             // Die Fehlerhaftigkeit des erkannten Parameter in der Fehlernummer eintragen   
             IF #piCount = 1 THEN
               #swParaError := #swParaError OR W#16#01;
             ELSIF #piCount = 2 THEN
               #swParaError := #swParaError OR W#16#02;
             ELSIF #piCount = 3 THEN
               #swParaError := #swParaError OR W#16#04;
             ELSIF #piCount = 4 THEN
               #swParaError := #swParaError OR W#16#08;
             ELSIF #piCount = 5 THEN
               #swParaError := #swParaError OR W#16#10;
             ELSIF #piCount = 6 THEN
               #swParaError := #swParaError OR W#16#20;
             ELSIF #piCount = 7 THEN
               #swParaError := #swParaError OR W#16#40;
             ELSIF #piCount = 8 THEN
               #swParaError := #swParaError OR W#16#80;
             ELSIF #piCount = 9 THEN
               #swParaError := #swParaError OR W#16#100;
             ELSIF #piCount = 10 THEN
               #swParaError := #swParaError OR W#16#200;
             ELSIF #piCount = 11 THEN
               #swParaError := #swParaError OR W#16#400;
             ELSIF #piCount = 12 THEN
               #swParaError := #swParaError OR W#16#800;
             ELSIF #piCount = 13 THEN
               #swParaError := #swParaError OR W#16#1000;
             ELSIF #piCount = 14 THEN
               #swParaError := #swParaError OR W#16#2000;
             ELSIF #piCount = 15 THEN
               #swParaError := #swParaError OR W#16#4000;
             ELSIF #piCount = #siParaNo THEN
               #swParaError := #swParaError OR W#16#8000;
             END_IF;

             // Zeiger auf nächsten Parametersatz setzen
             #piPointer := #piPointer + 6;

             // Format = Byte ? = > gesendeter Parameter ein Byte lang ohne Vorzeichen
           ELSIF (#sxRespParaMulti.sxData[#piPointer] = B#16#41) OR (#sxRespParaMulti.sxData[#piPointer] = B#16#05) THEN

             // ermittelter Parameterwert eintragen (Byte) 
             #sxParameter[#piCount].srValue := USINT_TO_REAL(BYTE_TO_USINT(#sxRespParaMulti.sxData[#piPointer + 2]));
             #sxParameter[#piCount].sdValue := 0;

             // ermittelte Fehlernummer im Puffer zurücksetzen
             #sxParameter[#piCount].swErrorNo := W#16#00;

             // Die Fehlerhaftigkeit des erkannten Parameter in der Fehlernummer löschen   
             IF #piCount = 1 THEN
               #swParaError := #swParaError AND W#16#FFFE;
             ELSIF #piCount = 2 THEN
               #swParaError := #swParaError AND W#16#FFFD;
             ELSIF #piCount = 3 THEN
               #swParaError := #swParaError AND W#16#FFFB;
             ELSIF #piCount = 4 THEN
               #swParaError := #swParaError AND W#16#FFF7;
             ELSIF #piCount = 5 THEN
               #swParaError := #swParaError AND W#16#FFEF;
             ELSIF #piCount = 6 THEN
               #swParaError := #swParaError AND W#16#FFDF;
             ELSIF #piCount = 7 THEN
               #swParaError := #swParaError AND W#16#FFBF;
             ELSIF #piCount = 8 THEN
               #swParaError := #swParaError AND W#16#FF7F;
             ELSIF #piCount = 9 THEN
               #swParaError := #swParaError AND W#16#FEFF;
             ELSIF #piCount = 10 THEN
               #swParaError := #swParaError AND W#16#FDFF;
             ELSIF #piCount = 11 THEN
               #swParaError := #swParaError AND W#16#FBFF;
             ELSIF #piCount = 12 THEN
               #swParaError := #swParaError AND W#16#F7FF;
             ELSIF #piCount = 13 THEN
               #swParaError := #swParaError AND W#16#EFFF;
             ELSIF #piCount = 14 THEN
               #swParaError := #swParaError AND W#16#DFFF;
             ELSIF #piCount = 15 THEN
               #swParaError := #swParaError AND W#16#BFFF;
             ELSIF #piCount = #siParaNo THEN
               #swParaError := #swParaError AND W#16#7FFF;
             END_IF;

             // Zeiger auf nächsten Parametersatz setzen
             #piPointer := #piPointer + 4;

             // Format = Byte ? = > gesendeter Parameter ein Byte lang mit Vorzeichen
           ELSIF (#sxRespParaMulti.sxData[#piPointer] = B#16#02) THEN

             // ermittelter Parameterwert eintragen (Byte) 
             #sxParameter[#piCount].srValue := SINT_TO_REAL(BYTE_TO_SINT(#sxRespParaMulti.sxData[#piPointer + 2]));
             #sxParameter[#piCount].sdValue := 0;

             // ermittelte Fehlernummer im Puffer zurücksetzen
             #sxParameter[#piCount].swErrorNo := W#16#00;

             // Die Fehlerhaftigkeit des erkannten Parameter in der Fehlernummer löschen   
             IF #piCount = 1 THEN
               #swParaError := #swParaError AND W#16#FFFE;
             ELSIF #piCount = 2 THEN
               #swParaError := #swParaError AND W#16#FFFD;
             ELSIF #piCount = 3 THEN
               #swParaError := #swParaError AND W#16#FFFB;
             ELSIF #piCount = 4 THEN
               #swParaError := #swParaError AND W#16#FFF7;
             ELSIF #piCount = 5 THEN
               #swParaError := #swParaError AND W#16#FFEF;
             ELSIF #piCount = 6 THEN
               #swParaError := #swParaError AND W#16#FFDF;
             ELSIF #piCount = 7 THEN
               #swParaError := #swParaError AND W#16#FFBF;
             ELSIF #piCount = 8 THEN
               #swParaError := #swParaError AND W#16#FF7F;
             ELSIF #piCount = 9 THEN
               #swParaError := #swParaError AND W#16#FEFF;
             ELSIF #piCount = 10 THEN
               #swParaError := #swParaError AND W#16#FDFF;
             ELSIF #piCount = 11 THEN
               #swParaError := #swParaError AND W#16#FBFF;
             ELSIF #piCount = 12 THEN
               #swParaError := #swParaError AND W#16#F7FF;
             ELSIF #piCount = 13 THEN
               #swParaError := #swParaError AND W#16#EFFF;
             ELSIF #piCount = 14 THEN
               #swParaError := #swParaError AND W#16#DFFF;
             ELSIF #piCount = 15 THEN
               #swParaError := #swParaError AND W#16#BFFF;
             ELSIF #piCount = #siParaNo THEN
               #swParaError := #swParaError AND W#16#7FFF;
             END_IF;

             // Zeiger auf nächsten Parametersatz setzen
             #piPointer := #piPointer + 4;

             // Format = Word ? = > gesendeter Parameter zwei Bytes lang ohne Vorzeichen
           ELSIF (#sxRespParaMulti.sxData[#piPointer] = B#16#42) OR (#sxRespParaMulti.sxData[#piPointer] = B#16#06)
             OR (#sxRespParaMulti.sxData[#piPointer] = B#16#0A) THEN

             // Format = Word, zwei Bytes zu übermitteltem Parameterwert zusammenfassen
             #pwWordHigh := SHL(IN := BYTE_TO_WORD(#sxRespParaMulti.sxData[#piPointer + 2]), N := 8);
             #pwWordLow := BYTE_TO_WORD(#sxRespParaMulti.sxData[#piPointer + 3]);
             #pwWord1 := #pwWordHigh XOR #pwWordLow;

             // ermittelter Parameterwert eintragen (Word)
             #sxParameter[#piCount].srValue := UINT_TO_REAL(WORD_TO_UINT(#pwWord1));
             #sxParameter[#piCount].sdValue := 0;

             // ermittelte Fehlernummer im Puffer zurücksetzen
             #sxParameter[#piCount].swErrorNo := W#16#00;

             // Die Fehlerhaftigkeit des erkannten Parameter in der Fehlernummer löschen   
             IF #piCount = 1 THEN
               #swParaError := #swParaError AND W#16#FFFE;
             ELSIF #piCount = 2 THEN
               #swParaError := #swParaError AND W#16#FFFD;
             ELSIF #piCount = 3 THEN
               #swParaError := #swParaError AND W#16#FFFB;
             ELSIF #piCount = 4 THEN
               #swParaError := #swParaError AND W#16#FFF7;
             ELSIF #piCount = 5 THEN
               #swParaError := #swParaError AND W#16#FFEF;
             ELSIF #piCount = 6 THEN
               #swParaError := #swParaError AND W#16#FFDF;
             ELSIF #piCount = 7 THEN
               #swParaError := #swParaError AND W#16#FFBF;
             ELSIF #piCount = 8 THEN
               #swParaError := #swParaError AND W#16#FF7F;
             ELSIF #piCount = 9 THEN
               #swParaError := #swParaError AND W#16#FEFF;
             ELSIF #piCount = 10 THEN
               #swParaError := #swParaError AND W#16#FDFF;
             ELSIF #piCount = 11 THEN
               #swParaError := #swParaError AND W#16#FBFF;
             ELSIF #piCount = 12 THEN
               #swParaError := #swParaError AND W#16#F7FF;
             ELSIF #piCount = 13 THEN
               #swParaError := #swParaError AND W#16#EFFF;
             ELSIF #piCount = 14 THEN
               #swParaError := #swParaError AND W#16#DFFF;
             ELSIF #piCount = 15 THEN
               #swParaError := #swParaError AND W#16#BFFF;
             ELSIF #piCount = #siParaNo THEN
               #swParaError := #swParaError AND W#16#7FFF;
             END_IF;

             // Zeiger auf nächsten Parametersatz setzen
             #piPointer := #piPointer + 4;

             // Format = Word ? = > gesendeter Parameter zwei Bytes lang mit Vorzeichen
           ELSIF (#sxRespParaMulti.sxData[#piPointer] = B#16#03) THEN

             // Format = Word, zwei Bytes zu übermitteltem Parameterwert zusammenfassen
             #pwWordHigh := SHL(IN := BYTE_TO_WORD(#sxRespParaMulti.sxData[#piPointer + 2]), N := 8);
             #pwWordLow := BYTE_TO_WORD(#sxRespParaMulti.sxData[#piPointer + 3]);
             #pwWord1 := #pwWordHigh XOR #pwWordLow;

             // ermittelter Parameterwert eintragen (Word)
             #sxParameter[#piCount].srValue := INT_TO_REAL(WORD_TO_INT(#pwWord1));
             #sxParameter[#piCount].sdValue := 0;

             // ermittelte Fehlernummer im Puffer zurücksetzen
             #sxParameter[#piCount].swErrorNo := W#16#00;

             // Die Fehlerhaftigkeit des erkannten Parameter in der Fehlernummer löschen   
             IF #piCount = 1 THEN
               #swParaError := #swParaError AND W#16#FFFE;
             ELSIF #piCount = 2 THEN
               #swParaError := #swParaError AND W#16#FFFD;
             ELSIF #piCount = 3 THEN
               #swParaError := #swParaError AND W#16#FFFB;
             ELSIF #piCount = 4 THEN
               #swParaError := #swParaError AND W#16#FFF7;
             ELSIF #piCount = 5 THEN
               #swParaError := #swParaError AND W#16#FFEF;
             ELSIF #piCount = 6 THEN
               #swParaError := #swParaError AND W#16#FFDF;
             ELSIF #piCount = 7 THEN
               #swParaError := #swParaError AND W#16#FFBF;
             ELSIF #piCount = 8 THEN
               #swParaError := #swParaError AND W#16#FF7F;
             ELSIF #piCount = 9 THEN
               #swParaError := #swParaError AND W#16#FEFF;
             ELSIF #piCount = 10 THEN
               #swParaError := #swParaError AND W#16#FDFF;
             ELSIF #piCount = 11 THEN
               #swParaError := #swParaError AND W#16#FBFF;
             ELSIF #piCount = 12 THEN
               #swParaError := #swParaError AND W#16#F7FF;
             ELSIF #piCount = 13 THEN
               #swParaError := #swParaError AND W#16#EFFF;
             ELSIF #piCount = 14 THEN
               #swParaError := #swParaError AND W#16#DFFF;
             ELSIF #piCount = 15 THEN
               #swParaError := #swParaError AND W#16#BFFF;
             ELSIF #piCount = #siParaNo THEN
               #swParaError := #swParaError AND W#16#7FFF;
             END_IF;

             // Zeiger auf nächsten Parametersatz setzen
             #piPointer := #piPointer + 4;

             // Format = Double Word ? = > gesendeter Parameter vier Bytes lang ohne Vorzeichen
           ELSIF (#sxRespParaMulti.sxData[#piPointer] = B#16#43) OR (#sxRespParaMulti.sxData[#piPointer] = B#16#07) OR
             (#sxRespParaMulti.sxData[#piPointer] = B#16#0D) THEN

             // Format = Double Word, vier Bytes zu übermitteltem Parameterwert zusammenfassen
             #pwWordHigh := SHL(IN := BYTE_TO_WORD(#sxRespParaMulti.sxData[#piPointer + 2]), N := 8);
             #pwWordLow := BYTE_TO_WORD(#sxRespParaMulti.sxData[#piPointer + 3]);
             #pwWord1 := #pwWordHigh XOR #pwWordLow;

             #pwWordHigh := SHL(IN := BYTE_TO_WORD(#sxRespParaMulti.sxData[#piPointer + 4]), N := 8);
             #pwWordLow := BYTE_TO_WORD(#sxRespParaMulti.sxData[#piPointer + 5]);
             #pwWord2 := #pwWordHigh XOR #pwWordLow;

             #pdDWordHigh := SHL(IN := WORD_TO_DWORD(#pwWord1), N := 16);
             #pdDWordLow := WORD_TO_DWORD(#pwWord2);

             // ermittelter Parameterwert eintragen (Word)
             #sxParameter[#piCount].srValue := 0.0;
             #sxParameter[#piCount].sdValue := DWORD_TO_DINT(#pdDWordHigh XOR #pdDWordLow);

             // ermittelte Fehlernummer im Puffer zurücksetzen
             #sxParameter[#piCount].swErrorNo := W#16#00;

             // Die Fehlerhaftigkeit des erkannten Parameter in der Fehlernummer löschen   
             IF #piCount = 1 THEN
               #swParaError := #swParaError AND W#16#FFFE;
             ELSIF #piCount = 2 THEN
               #swParaError := #swParaError AND W#16#FFFD;
             ELSIF #piCount = 3 THEN
               #swParaError := #swParaError AND W#16#FFFB;
             ELSIF #piCount = 4 THEN
               #swParaError := #swParaError AND W#16#FFF7;
             ELSIF #piCount = 5 THEN
               #swParaError := #swParaError AND W#16#FFEF;
             ELSIF #piCount = 6 THEN
               #swParaError := #swParaError AND W#16#FFDF;
             ELSIF #piCount = 7 THEN
               #swParaError := #swParaError AND W#16#FFBF;
             ELSIF #piCount = 8 THEN
               #swParaError := #swParaError AND W#16#FF7F;
             ELSIF #piCount = 9 THEN
               #swParaError := #swParaError AND W#16#FEFF;
             ELSIF #piCount = 10 THEN
               #swParaError := #swParaError AND W#16#FDFF;
             ELSIF #piCount = 11 THEN
               #swParaError := #swParaError AND W#16#FBFF;
             ELSIF #piCount = 12 THEN
               #swParaError := #swParaError AND W#16#F7FF;
             ELSIF #piCount = 13 THEN
               #swParaError := #swParaError AND W#16#EFFF;
             ELSIF #piCount = 14 THEN
               #swParaError := #swParaError AND W#16#DFFF;
             ELSIF #piCount = 15 THEN
               #swParaError := #swParaError AND W#16#BFFF;
             ELSIF #piCount = #siParaNo THEN
               #swParaError := #swParaError AND W#16#7FFF;
             END_IF;

             // Zeiger auf nächsten Parametersatz setzen
             #piPointer := #piPointer + 6;

             // Format = Double Word ? = > gesendeter Parameter vier Bytes lang mit Vorzeichen
           ELSIF (#sxRespParaMulti.sxData[#piPointer] = B#16#04) THEN

             // Format = Double Word, vier Bytes zu übermitteltem Parameterwert zusammenfassen
             #pwWordHigh := SHL(IN := BYTE_TO_WORD(#sxRespParaMulti.sxData[#piPointer + 2]), N := 8);
             #pwWordLow := BYTE_TO_WORD(#sxRespParaMulti.sxData[#piPointer + 3]);
             #pwWord1 := #pwWordHigh XOR #pwWordLow;

             #pwWordHigh := SHL(IN := BYTE_TO_WORD(#sxRespParaMulti.sxData[#piPointer + 4]), N := 8);
             #pwWordLow := BYTE_TO_WORD(#sxRespParaMulti.sxData[#piPointer + 5]);
             #pwWord2 := #pwWordHigh XOR #pwWordLow;

             #pdDWordHigh := SHL(IN := WORD_TO_DWORD(#pwWord1), N := 16);
             #pdDWordLow := WORD_TO_DWORD(#pwWord2);

             // ermittelter Parameterwert eintragen (Word)
             #sxParameter[#piCount].srValue := 0.0;
             #sxParameter[#piCount].sdValue := DWORD_TO_DINT(#pdDWordHigh XOR #pdDWordLow);

             // ermittelte Fehlernummer im Puffer zurücksetzen
             #sxParameter[#piCount].swErrorNo := W#16#00;

             // Die Fehlerhaftigkeit des erkannten Parameter in der Fehlernummer löschen   
             IF #piCount = 1 THEN
               #swParaError := #swParaError AND W#16#FFFE;
             ELSIF #piCount = 2 THEN
               #swParaError := #swParaError AND W#16#FFFD;
             ELSIF #piCount = 3 THEN
               #swParaError := #swParaError AND W#16#FFFB;
             ELSIF #piCount = 4 THEN
               #swParaError := #swParaError AND W#16#FFF7;
             ELSIF #piCount = 5 THEN
               #swParaError := #swParaError AND W#16#FFEF;
             ELSIF #piCount = 6 THEN
               #swParaError := #swParaError AND W#16#FFDF;
             ELSIF #piCount = 7 THEN
               #swParaError := #swParaError AND W#16#FFBF;
             ELSIF #piCount = 8 THEN
               #swParaError := #swParaError AND W#16#FF7F;
             ELSIF #piCount = 9 THEN
               #swParaError := #swParaError AND W#16#FEFF;
             ELSIF #piCount = 10 THEN
               #swParaError := #swParaError AND W#16#FDFF;
             ELSIF #piCount = 11 THEN
               #swParaError := #swParaError AND W#16#FBFF;
             ELSIF #piCount = 12 THEN
               #swParaError := #swParaError AND W#16#F7FF;
             ELSIF #piCount = 13 THEN
               #swParaError := #swParaError AND W#16#EFFF;
             ELSIF #piCount = 14 THEN
               #swParaError := #swParaError AND W#16#DFFF;
             ELSIF #piCount = 15 THEN
               #swParaError := #swParaError AND W#16#BFFF;
             ELSIF #piCount = #siParaNo THEN
               #swParaError := #swParaError AND W#16#7FFF;
             END_IF;

             // Zeiger auf nächsten Parametersatz setzen
             #piPointer := #piPointer + 6;

             // Format = Double Word ? = > gesendeter Parameter vier Bytes lang (FloatingPoint)
           ELSIF (#sxRespParaMulti.sxData[#piPointer] = B#16#08) THEN

             // Format = Double Word, vier Bytes zu übermitteltem Parameterwert zusammenfassen
             #pwWordHigh := SHL(IN := BYTE_TO_WORD(#sxRespParaMulti.sxData[#piPointer + 2]), N := 8);
             #pwWordLow := BYTE_TO_WORD(#sxRespParaMulti.sxData[#piPointer + 3]);
             #pwWord1 := #pwWordHigh XOR #pwWordLow;

             #pwWordHigh := SHL(IN := BYTE_TO_WORD(#sxRespParaMulti.sxData[#piPointer + 4]), N := 8);
             #pwWordLow := BYTE_TO_WORD(#sxRespParaMulti.sxData[#piPointer + 5]);
             #pwWord2 := #pwWordHigh XOR #pwWordLow;

             #pdDWordHigh := SHL(IN := WORD_TO_DWORD(#pwWord1), N := 16);
             #pdDWordLow := WORD_TO_DWORD(#pwWord2);

             // ermittelter Parameterwert eintragen (Word)
             #sxParameter[#piCount].srValue := DWORD_TO_REAL(#pdDWordHigh XOR #pdDWordLow);
             #sxParameter[#piCount].sdValue := 0;

             // ermittelte Fehlernummer im Puffer zurücksetzen
             #sxParameter[#piCount].swErrorNo := W#16#00;

             // Die Fehlerhaftigkeit des erkannten Parameter in der Fehlernummer löschen   
             IF #piCount = 1 THEN
               #swParaError := #swParaError AND W#16#FFFE;
             ELSIF #piCount = 2 THEN
               #swParaError := #swParaError AND W#16#FFFD;
             ELSIF #piCount = 3 THEN
               #swParaError := #swParaError AND W#16#FFFB;
             ELSIF #piCount = 4 THEN
               #swParaError := #swParaError AND W#16#FFF7;
             ELSIF #piCount = 5 THEN
               #swParaError := #swParaError AND W#16#FFEF;
             ELSIF #piCount = 6 THEN
               #swParaError := #swParaError AND W#16#FFDF;
             ELSIF #piCount = 7 THEN
               #swParaError := #swParaError AND W#16#FFBF;
             ELSIF #piCount = 8 THEN
               #swParaError := #swParaError AND W#16#FF7F;
             ELSIF #piCount = 9 THEN
               #swParaError := #swParaError AND W#16#FEFF;
             ELSIF #piCount = 10 THEN
               #swParaError := #swParaError AND W#16#FDFF;
             ELSIF #piCount = 11 THEN
               #swParaError := #swParaError AND W#16#FBFF;
             ELSIF #piCount = 12 THEN
               #swParaError := #swParaError AND W#16#F7FF;
             ELSIF #piCount = 13 THEN
               #swParaError := #swParaError AND W#16#EFFF;
             ELSIF #piCount = 14 THEN
               #swParaError := #swParaError AND W#16#DFFF;
             ELSIF #piCount = 15 THEN
               #swParaError := #swParaError AND W#16#BFFF;
             ELSIF #piCount = #siParaNo THEN
               #swParaError := #swParaError AND W#16#7FFF;
             END_IF;

             // Zeiger auf nächsten Parametersatz setzen
             #piPointer := #piPointer + 6;

             // Unbekanter Datentyp
           ELSE

             #siErrorId := 5;
             #sbError := True;
             #sbDone := False;
             // Die Fehlerhaftigkeit des erkannten Parameter in der Fehlernummer eintragen   
             IF #piCount = 1 THEN
               #swParaError := #swParaError OR W#16#01;
             ELSIF #piCount = 2 THEN
               #swParaError := #swParaError OR W#16#02;
             ELSIF #piCount = 3 THEN
               #swParaError := #swParaError OR W#16#04;
             ELSIF #piCount = 4 THEN
               #swParaError := #swParaError OR W#16#08;
             ELSIF #piCount = 5 THEN
               #swParaError := #swParaError OR W#16#10;
             ELSIF #piCount = 6 THEN
               #swParaError := #swParaError OR W#16#20;
             ELSIF #piCount = 7 THEN
               #swParaError := #swParaError OR W#16#40;
             ELSIF #piCount = 8 THEN
               #swParaError := #swParaError OR W#16#80;
             ELSIF #piCount = 9 THEN
               #swParaError := #swParaError OR W#16#100;
             ELSIF #piCount = 10 THEN
               #swParaError := #swParaError OR W#16#200;
             ELSIF #piCount = 11 THEN
               #swParaError := #swParaError OR W#16#400;
             ELSIF #piCount = 12 THEN
               #swParaError := #swParaError OR W#16#800;
             ELSIF #piCount = 13 THEN
               #swParaError := #swParaError OR W#16#1000;
             ELSIF #piCount = 14 THEN
               #swParaError := #swParaError OR W#16#2000;
             ELSIF #piCount = 15 THEN
               #swParaError := #swParaError OR W#16#4000;
             ELSIF #piCount = #siParaNo THEN
               #swParaError := #swParaError OR W#16#8000;
             END_IF;

             EXIT; //Bei erstem unbekannten Datentyp abrechen

           END_IF;
         END_FOR; // die angefragten Parameter auswerten und im Puffer abspeichern

         // Fehlerkennung zurücknehmen
         IF (#siErrorId = 3) OR (#siErrorId = 1) THEN
           #siErrorId := 0;
           #sbError := False;
         END_IF;

         #DiagId := W#16#00;

         // Auftrag : Parameter lesen ist abgeschlossen
         #sbRdStart := False;
         #sbRead := False;
       END_IF; // kein Fehler beim LESEN AZYKLISCH und Auftrag fertig 
     END_IF; // vom Auftrag "Parameter lesen" die Antwort abwarten und dann auswerten
   END_IF; // Auftrag "Parameter lesen" wurde ausgelöst


   // Auftrag "Parameter schreiben" wurde ausgelöst
   IF #sbParaNo AND NOT #sbRead AND #sbWrite THEN

     // Auftrag "Parameter schreiben" bzw. "ändern" besteht aus zwei Aufträgen
     // 1. Teilauftrag "Parameter lesen"
     // 2. Teilauftrag "Parameter schreiben bzw. ändern"

     // 1. Teilauftrag "Parameter lesen" vorbereiten und abschicken
     IF #sbWrStart1 THEN

       // Ablöschen des Sendepuffers
       IF NOT (#siParaNo = #siParaNoMax) THEN
         FOR #piCount := #siParaNo TO #siParaNoMax DO

           // Parameternummer des Parameters 
           #sxReqParaMulti.sxParaAdress[#piCount].siParaNo := 0;

           // Subindex des Parameters
           #sxReqParaMulti.sxParaAdress[#piCount].siIndex := 0;
         END_FOR;
       END_IF;

       // Auftrags-HEADER erstellen
       // Auftragsreferenz
       #sxReqParaMulti.sxHeader.syReqRef := INT_TO_BYTE(#siReqRef);

       // Auftragskennung 0x01=Request Parameters
       #sxReqParaMulti.sxHeader.syReqId := B#16#01;

       // Achse
       #sxReqParaMulti.sxHeader.syAxisNo := #syAxisNo;

       // Anzahl Parameter        
       #sxReqParaMulti.sxHeader.syParaNo := INT_TO_BYTE(#siParaNo);

       // Auftrags-PARAMETERADRESSE erstellen
       FOR #piCount := 1 TO #siParaNo DO

         // Parameternummer des Parameters                                
         #sxReqParaMulti.sxParaAdress[#piCount].siParaNo := #sxParameter[#piCount].siParaNo;

         // Subindex des Parameters
         #sxReqParaMulti.sxParaAdress[#piCount].siIndex := #sxParameter[#piCount].siIndex;
       END_FOR;

       // SCHREIBEN AZYKLISCH
       #piLenTele := #siLenHeader + #siLenParaMulti;
       #WRREC_1(REQ := True,                                // Startimpuls
                ID := #hardwareId,                         // Diagnoseadresse
                INDEX := 47,                                  // Rahmentyp
                LEN := INT_TO_UINT(#piLenTele),             // maximale Länge
                DONE => #sbWrDone,                           // Schreibauftrag beendet
                BUSY => #sbWrBusy,                           // Slave beschäftigt
                ERROR => #sbWrError,                          // Fehler beim Schreiben
                STATUS => #pdStatus,                           // Status[1] = Error => Status[2] Error Decode + Status[3] Error Code
                RECORD := #sxReqParaMulti);                    // Zeiger auf zu schreibenen Datensatz

       // Ausgänge setzen
       #sbBusy := #sbWrBusy;
       #sbDone := #sbWrDone;

       // Fehler auswerten
       IF #sbWrError THEN

         // Fehlerstatus aus dem Doppelwort filtern und weitergeben                
         #pwWord1 := DWORD_TO_WORD(SHR(IN := (#pdStatus AND DW#16#FFFF00), N := 8));

         // Fehlerstatus setzen
         #siErrorId := 3;
         #DiagId := #pwWord1;

         //Temporärer Fehler: #pdStatus = 80A7, 80B5, 80C0, 80C1, 80C2, 80C3 oder 80C4 zulassen und nocheinmal versuchen
         IF NOT (#pwWord1 = DW#16#80A7) AND NOT (#pwWord1 = DW#16#80B5) AND NOT (#pwWord1 = DW#16#80C0) AND
           NOT (#pwWord1 = DW#16#80C1) AND NOT (#pwWord1 = DW#16#80C2) AND NOT (#pwWord1 = DW#16#80C3) AND
           NOT (#pwWord1 = DW#16#80C4) THEN

           // Wiederholungsauftrag wieder zurücknehmen
           #sbWrStart1 := False;
           #sbRdStart1 := False;
           #sbWrite := False;

           // Fehler ausgeben 
           #sbError := #sbWrError;

         ELSE
           // Fehlerwiederholauftrag ??                   
           IF #siErrorCount = #siMaxErrCount THEN

             // Wiederholungsauftrag wieder zurücknehmen
             #sbWrStart1 := False;
             #sbRdStart1 := False;
             #sbWrite := False;

             //Fehlerzähler zurücksetzen
             #siErrorCount := 0;

             // Fehler ausgeben 
             #sbError := #sbWrError;

             // nix tun bis Zähler überläuft
           ELSE
             #siErrorCount := #siErrorCount + 1;
           END_IF;
         END_IF;

         // kein Fehler beim SCHEIBEN AZYKLISCH und Auftrag fertig 
       ELSIF NOT #sbWrBusy AND #sbWrDone THEN

         // Fehlerkennung zurücknehmen
         IF (#siErrorId = 3) THEN
           #siErrorId := 0;
           #sbError := False;
         END_IF;

         #DiagId := W#16#00;

         // Schreibauftrag fertig melden und Leseantrag anstossen
         #sbWrStart1 := False;
         #sbRdStart1 := True;
       END_IF;
     END_IF; // 1. Teilauftrag "Parameter lesen" vorbereiten und abschicken

     // vom 1. Teilauftrag "Parameter lesen" die Antwort abwarten und dann auswerten
     IF #sbRdStart1 THEN

       // Ablöschen des Empfangspuffers
       #sxRespParaMulti.sxHeader.syReqRef := B#16#00;
       #sxRespParaMulti.sxHeader.syReqId := B#16#00;
       #sxRespParaMulti.sxHeader.syAxisNo := B#16#00;
       #sxRespParaMulti.sxHeader.syParaNo := B#16#00;

       FOR #piCount := 1 TO #siLenParaMulti DO
         #sxRespParaMulti.sxData[#piCount] := B#16#00;
       END_FOR;

       // LESEN AZYKLISCH
       #piLenTele := #siLenHeader + #siLenParaMulti;
       #RDREC_1(REQ := True,                                // Startimpuls
                ID := #hardwareId,                         // Diagnoseadresse        
                INDEX := 47,                                  // Rahmentyp           
                MLEN := INT_TO_UINT(#piLenTele),             // maximale Länge
                VALID => #pbValidSFB,                         // neuer Datensatz empfangen und gültig      
                BUSY => #sbRdBusy,                           // Slave beschäftigt
                ERROR => #sbRdError,                          // Fehler beim Schreiben
                STATUS => #pdStatus,                           // Status[1] = Error => Status[2] Error Decode + Status[3] Error Code 
                LEN => #piLenSFB,                           // Länge des gelesenen Datensatzes
                RECORD := #sxRespParaMulti);                   // Zeiger auf gelesenen Datensatz

       // Ausgänge setzen
       #sbBusy := #sbRdBusy;
       #sbDone := #pbValidSFB;

       // Fehler auswerten
       IF #sbRdError THEN
         // Fehlerstatus aus dem Doppelwort filtern und weitergeben                
         #pwWord1 := DWORD_TO_WORD(SHR(IN := (#pdStatus AND DW#16#FFFF00), N := 8));

         // Fehlerstatus setzen
         #siErrorId := 3;
         #DiagId := #pwWord1;

         //Temporärer Fehler: #pdStatus = 80A7, 80B5, 80C0, 80C1, 80C2, 80C3 oder 80C4 zulassen und nocheinmal versuchen
         IF NOT (#pwWord1 = DW#16#80A7) AND NOT (#pwWord1 = DW#16#80B5) AND NOT (#pwWord1 = DW#16#80C0) AND
           NOT (#pwWord1 = DW#16#80C1) AND NOT (#pwWord1 = DW#16#80C2) AND NOT (#pwWord1 = DW#16#80C3) AND
           NOT (#pwWord1 = DW#16#80C4) THEN

           // Wiederholungsauftrag wieder zurücknehmen
           #sbWrStart1 := False;
           #sbRdStart1 := False;
           #sbWrite := False;

           // Fehler ausgeben 
           #sbError := #sbRdError;

         ELSE
           // Fehlerwiederholauftrag ??                   
           IF #siErrorCount = #siMaxErrCount THEN

             // Wiederholungsauftrag wieder zurücknehmen
             #sbWrStart1 := False;
             #sbRdStart1 := False;
             #sbWrite := False;

             //Fehlerzähler zurücksetzen
             #siErrorCount := 0;

             // Fehler ausgeben 
             #sbError := #sbRdError;

             // nix tun bis Zähler überläuft
           ELSE
             #siErrorCount := #siErrorCount + 1;
           END_IF;
         END_IF;

         // Fehler : die Auftragsreferenz der Antwort übertimmt nicht mit der Auftragsreferenz der Anfrage überein
       ELSIF NOT (#siReqRef = BYTE_TO_INT(#sxRespParaMulti.sxHeader.syReqRef)) AND NOT #sbRdBusy AND #pbValidSFB THEN
         #siErrorId := 1;
         #sbError := True;
         #sbDone := False;

         // Wiederholungsauftrag wieder zurücknehmen
         #sbWrStart1 := False;
         #sbRdStart1 := False;
         #sbWrite := False;

         // Fehler : falsche Auftragskennung zurück erhalten    
       ELSIF NOT (#sxRespParaMulti.sxHeader.syReqId = B#16#81 OR #sxRespParaMulti.sxHeader.syReqId = B#16#01) AND
         NOT #sbRdBusy AND #pbValidSFB THEN
         #siErrorId := 1;
         #sbError := True;
         #sbDone := False;

         // Wiederholungsauftrag wieder zurücknehmen
         #sbWrStart1 := False;
         #sbRdStart1 := False;
         #sbWrite := False;

         // Fehler : die angeforderte Anzahl Parameter entspricht nicht der übermittelten Anzahl Parameter überein
       ELSIF NOT (#siParaNo = BYTE_TO_INT(#sxRespParaMulti.sxHeader.syParaNo)) AND NOT #sbRdBusy AND #pbValidSFB THEN
         #siErrorId := 1;
         #sbError := True;
         #sbDone := False;

         // Wiederholungsauftrag wieder zurücknehmen
         #sbWrStart1 := False;
         #sbRdStart1 := False;
         #sbWrite := False;

         // Fehler : die Achse entspricht nicht der übergebenen Achse
       ELSIF NOT (#syAxisNo = #sxRespParaMulti.sxHeader.syAxisNo) AND NOT #sbRdBusy AND #pbValidSFB THEN
         #siErrorId := 1;
         #sbError := True;
         #sbDone := False;

         // Wiederholungsauftrag wieder zurücknehmen
         #sbWrStart1 := False;
         #sbRdStart1 := False;
         #sbWrite := False;

         // kein Fehler beim LESEN AZYKLISCH und Auftrag fertig 
       ELSIF NOT #sbRdBusy AND #pbValidSFB THEN

         // die angefragten Parameter auswerten und im Puffer abspeichern
         #piPointer := 1;
         #swParaError := 16#0;

         FOR #piCount := 1 TO #siParaNo DO

           // ermitteltes Format des Parameters abspeichern
           #sxParameter[#piCount].syFormat := #sxRespParaMulti.sxData[#piPointer];

           // Format = Error ? = > gesendeter Parameter fehlerhaft
           IF (BYTE_TO_INT(#sxRespParaMulti.sxData[#piPointer]) = 68) THEN

             // Format = Error, zwei Bytes zu übermittelten Fehlernummer zusammenfassen
             #pwWordHigh := SHL(IN := BYTE_TO_WORD(#sxRespParaMulti.sxData[#piPointer + 2]), N := 8);
             #pwWordLow := BYTE_TO_WORD(#sxRespParaMulti.sxData[#piPointer + 3]);

             #sbError := True;

             // ermittelte Fehlernummer im Puffer abspeichern
             #sxParameter[#piCount].swErrorNo := #pwWordHigh XOR #pwWordLow;

             // Die Fehlerhaftigkeit des erkannten Parameter in der Fehlernummer eintragen   
             IF #piCount = 1 THEN
               #swParaError := #swParaError OR W#16#01;
             ELSIF #piCount = 2 THEN
               #swParaError := #swParaError OR W#16#02;
             ELSIF #piCount = 3 THEN
               #swParaError := #swParaError OR W#16#04;
             ELSIF #piCount = 4 THEN
               #swParaError := #swParaError OR W#16#08;
             ELSIF #piCount = 5 THEN
               #swParaError := #swParaError OR W#16#10;
             ELSIF #piCount = 6 THEN
               #swParaError := #swParaError OR W#16#20;
             ELSIF #piCount = 7 THEN
               #swParaError := #swParaError OR W#16#40;
             ELSIF #piCount = 8 THEN
               #swParaError := #swParaError OR W#16#80;
             ELSIF #piCount = 9 THEN
               #swParaError := #swParaError OR W#16#100;
             ELSIF #piCount = 10 THEN
               #swParaError := #swParaError OR W#16#200;
             ELSIF #piCount = 11 THEN
               #swParaError := #swParaError OR W#16#400;
             ELSIF #piCount = 12 THEN
               #swParaError := #swParaError OR W#16#800;
             ELSIF #piCount = 13 THEN
               #swParaError := #swParaError OR W#16#1000;
             ELSIF #piCount = 14 THEN
               #swParaError := #swParaError OR W#16#2000;
             ELSIF #piCount = 15 THEN
               #swParaError := #swParaError OR W#16#4000;
             ELSIF #piCount = #siParaNo THEN
               #swParaError := #swParaError OR W#16#8000;
             END_IF;

             // Zeiger auf nächsten Parametersatz setzen
             #piPointer := #piPointer + 6;

             // Format = Byte ? = > gesendeter Parameter ein Byte lang
           ELSIF (#sxRespParaMulti.sxData[#piPointer] = B#16#41) OR
             (#sxRespParaMulti.sxData[#piPointer] = B#16#02) OR (#sxRespParaMulti.sxData[#piPointer] = B#16#05) THEN

             // ermittelte Fehlernummer im Puffer zurücksetzen
             #sxParameter[#piCount].swErrorNo := W#16#00;

             // Die Fehlerhaftigkeit des erkannten Parameter in der Fehlernummer löschen   
             IF #piCount = 1 THEN
               #swParaError := #swParaError AND W#16#FFFE;
             ELSIF #piCount = 2 THEN
               #swParaError := #swParaError AND W#16#FFFD;
             ELSIF #piCount = 3 THEN
               #swParaError := #swParaError AND W#16#FFFB;
             ELSIF #piCount = 4 THEN
               #swParaError := #swParaError AND W#16#FFF7;
             ELSIF #piCount = 5 THEN
               #swParaError := #swParaError AND W#16#FFEF;
             ELSIF #piCount = 6 THEN
               #swParaError := #swParaError AND W#16#FFDF;
             ELSIF #piCount = 7 THEN
               #swParaError := #swParaError AND W#16#FFBF;
             ELSIF #piCount = 8 THEN
               #swParaError := #swParaError AND W#16#FF7F;
             ELSIF #piCount = 9 THEN
               #swParaError := #swParaError AND W#16#FEFF;
             ELSIF #piCount = 10 THEN
               #swParaError := #swParaError AND W#16#FDFF;
             ELSIF #piCount = 11 THEN
               #swParaError := #swParaError AND W#16#FBFF;
             ELSIF #piCount = 12 THEN
               #swParaError := #swParaError AND W#16#F7FF;
             ELSIF #piCount = 13 THEN
               #swParaError := #swParaError AND W#16#EFFF;
             ELSIF #piCount = 14 THEN
               #swParaError := #swParaError AND W#16#DFFF;
             ELSIF #piCount = 15 THEN
               #swParaError := #swParaError AND W#16#BFFF;
             ELSIF #piCount = #siParaNo THEN
               #swParaError := #swParaError AND W#16#7FFF;
             END_IF;

             // Zeiger auf nächsten Parametersatz setzen
             #piPointer := #piPointer + 4;

             // Format = Word ? = > gesendeter Parameter zwei Bytes lang
           ELSIF (#sxRespParaMulti.sxData[#piPointer] = B#16#42) OR (#sxRespParaMulti.sxData[#piPointer] = B#16#03)
             OR (#sxRespParaMulti.sxData[#piPointer] = B#16#06) OR (#sxRespParaMulti.sxData[#piPointer] = B#16#0A) THEN

             // ermittelte Fehlernummer im Puffer zurücksetzen
             #sxParameter[#piCount].swErrorNo := W#16#00;

             // Die Fehlerhaftigkeit des erkannten Parameter in der Fehlernummer löschen   
             IF #piCount = 1 THEN
               #swParaError := #swParaError AND W#16#FFFE;
             ELSIF #piCount = 2 THEN
               #swParaError := #swParaError AND W#16#FFFD;
             ELSIF #piCount = 3 THEN
               #swParaError := #swParaError AND W#16#FFFB;
             ELSIF #piCount = 4 THEN
               #swParaError := #swParaError AND W#16#FFF7;
             ELSIF #piCount = 5 THEN
               #swParaError := #swParaError AND W#16#FFEF;
             ELSIF #piCount = 6 THEN
               #swParaError := #swParaError AND W#16#FFDF;
             ELSIF #piCount = 7 THEN
               #swParaError := #swParaError AND W#16#FFBF;
             ELSIF #piCount = 8 THEN
               #swParaError := #swParaError AND W#16#FF7F;
             ELSIF #piCount = 9 THEN
               #swParaError := #swParaError AND W#16#FEFF;
             ELSIF #piCount = 10 THEN
               #swParaError := #swParaError AND W#16#FDFF;
             ELSIF #piCount = 11 THEN
               #swParaError := #swParaError AND W#16#FBFF;
             ELSIF #piCount = 12 THEN
               #swParaError := #swParaError AND W#16#F7FF;
             ELSIF #piCount = 13 THEN
               #swParaError := #swParaError AND W#16#EFFF;
             ELSIF #piCount = 14 THEN
               #swParaError := #swParaError AND W#16#DFFF;
             ELSIF #piCount = 15 THEN
               #swParaError := #swParaError AND W#16#BFFF;
             ELSIF #piCount = #siParaNo THEN
               #swParaError := #swParaError AND W#16#7FFF;
             END_IF;

             // Zeiger auf nächsten Parametersatz setzen
             #piPointer := #piPointer + 4;

             // Format = Double Word ? = > gesendeter Parameter vier Bytes lang
           ELSIF (#sxRespParaMulti.sxData[#piPointer] = B#16#43) OR (#sxRespParaMulti.sxData[#piPointer] = B#16#04) OR
             (#sxRespParaMulti.sxData[#piPointer] = B#16#07) OR (#sxRespParaMulti.sxData[#piPointer] = B#16#08) OR
             (#sxRespParaMulti.sxData[#piPointer] = B#16#0D) THEN

             // ermittelte Fehlernummer im Puffer zurücksetzen
             #sxParameter[#piCount].swErrorNo := W#16#00;

             // Die Fehlerhaftigkeit des erkannten Parameter in der Fehlernummer löschen   
             IF #piCount = 1 THEN
               #swParaError := #swParaError AND W#16#FFFE;
             ELSIF #piCount = 2 THEN
               #swParaError := #swParaError AND W#16#FFFD;
             ELSIF #piCount = 3 THEN
               #swParaError := #swParaError AND W#16#FFFB;
             ELSIF #piCount = 4 THEN
               #swParaError := #swParaError AND W#16#FFF7;
             ELSIF #piCount = 5 THEN
               #swParaError := #swParaError AND W#16#FFEF;
             ELSIF #piCount = 6 THEN
               #swParaError := #swParaError AND W#16#FFDF;
             ELSIF #piCount = 7 THEN
               #swParaError := #swParaError AND W#16#FFBF;
             ELSIF #piCount = 8 THEN
               #swParaError := #swParaError AND W#16#FF7F;
             ELSIF #piCount = 9 THEN
               #swParaError := #swParaError AND W#16#FEFF;
             ELSIF #piCount = 10 THEN
               #swParaError := #swParaError AND W#16#FDFF;
             ELSIF #piCount = 11 THEN
               #swParaError := #swParaError AND W#16#FBFF;
             ELSIF #piCount = 12 THEN
               #swParaError := #swParaError AND W#16#F7FF;
             ELSIF #piCount = 13 THEN
               #swParaError := #swParaError AND W#16#EFFF;
             ELSIF #piCount = 14 THEN
               #swParaError := #swParaError AND W#16#DFFF;
             ELSIF #piCount = 15 THEN
               #swParaError := #swParaError AND W#16#BFFF;
             ELSIF #piCount = #siParaNo THEN
               #swParaError := #swParaError AND W#16#7FFF;
             END_IF;

             // Zeiger auf nächsten Parametersatz setzen
             #piPointer := #piPointer + 6;

             // Unbekanter Datentyp
           ELSE

             #siErrorId := 5;
             #sbError := True;
             #sbDone := False;
             // Die Fehlerhaftigkeit des erkannten Parameter in der Fehlernummer eintragen   
             IF #piCount = 1 THEN
               #swParaError := #swParaError OR W#16#01;
             ELSIF #piCount = 2 THEN
               #swParaError := #swParaError OR W#16#02;
             ELSIF #piCount = 3 THEN
               #swParaError := #swParaError OR W#16#04;
             ELSIF #piCount = 4 THEN
               #swParaError := #swParaError OR W#16#08;
             ELSIF #piCount = 5 THEN
               #swParaError := #swParaError OR W#16#10;
             ELSIF #piCount = 6 THEN
               #swParaError := #swParaError OR W#16#20;
             ELSIF #piCount = 7 THEN
               #swParaError := #swParaError OR W#16#40;
             ELSIF #piCount = 8 THEN
               #swParaError := #swParaError OR W#16#80;
             ELSIF #piCount = 9 THEN
               #swParaError := #swParaError OR W#16#100;
             ELSIF #piCount = 10 THEN
               #swParaError := #swParaError OR W#16#200;
             ELSIF #piCount = 11 THEN
               #swParaError := #swParaError OR W#16#400;
             ELSIF #piCount = 12 THEN
               #swParaError := #swParaError OR W#16#800;
             ELSIF #piCount = 13 THEN
               #swParaError := #swParaError OR W#16#1000;
             ELSIF #piCount = 14 THEN
               #swParaError := #swParaError OR W#16#2000;
             ELSIF #piCount = 15 THEN
               #swParaError := #swParaError OR W#16#4000;
             ELSIF #piCount = #siParaNo THEN
               #swParaError := #swParaError OR W#16#8000;
             END_IF;

             EXIT; //Bei erstem unbekannten Datentyp abrechen

           END_IF;
         END_FOR; // die angefragten Parameter auswerten und im Puffer abspeichern

         // Fehlerkennung zurücknehmen
         IF (#siErrorId = 3) OR (#siErrorId = 1) THEN
           #siErrorId := 0;
           #sbError := False;
         END_IF;

         #DiagId := W#16#00;

         // 1. Teilauftrag "Parameter lesen" ist abgeschlossen
         #sbRdStart1 := False;

         // einer der gesendeten Parameter ist fehlerhaft => Abbruch, kein "Parameter schreiben" erforderlich
         IF (#swParaError = W#16#00) THEN
           #sbWrStart2 := True;
         ELSE
           #sbWrStart2 := False;
         END_IF;
       END_IF; // kein Fehler beim LESEN AZYKLISCH und Auftrag fertig 
     END_IF; // vom 1. Teilauftrag "Parameter lesen" die Antwort abwarten und dann auswerten 

     // 2. Teilauftrag "Parameter schreiben bzw. ändern" vorbereiten und abschicken
     IF #sbWrStart2 THEN

       // Ablöschen des Sendepuffers            
       FOR #piCount := 1 TO #siLenChaPara DO
         // Parameteradresse und Parameterwert des Parameters 
         #sxChaParaMulti.sxData[#piCount] := B#16#00;
       END_FOR;

       // Auftrags-HEADER erstellen
       // Auftragsreferenz
       #sxChaParaMulti.sxHeader.syReqRef := INT_TO_BYTE(#siReqRef);

       // Auftragskennung 0x01=Request Parameters | 0x02=Change Parameters
       #sxChaParaMulti.sxHeader.syReqId := B#16#02;

       // Achse
       #sxChaParaMulti.sxHeader.syAxisNo := #syAxisNo;

       // Anzahl Parameter        
       #sxChaParaMulti.sxHeader.syParaNo := INT_TO_BYTE(#siParaNo);

       // Auftrags-PARAMETERADRESSE erstellen
       #piPointer := 1;
       FOR #piCount := 1 TO #siParaNo DO

         // Attribute of parameters (0x10=Value, 0x30=Text)
         #sxChaParaMulti.sxData[#piPointer] := B#16#10;

         // No. of elements (DEC: for single elements=1) 
         #sxChaParaMulti.sxData[#piPointer + 1] := B#16#01;

         // Parameternummer des Parameters                                
         #sxChaParaMulti.sxData[#piPointer + 3] := INT_TO_BYTE(#sxParameter[#piCount].siParaNo);
         #sxChaParaMulti.sxData[#piPointer + 2] := WORD_TO_BYTE(SHR(IN := INT_TO_WORD(#sxParameter[#piCount].siParaNo), N := 8));

         // Subindex des Parameters
         #sxChaParaMulti.sxData[#piPointer + 5] := INT_TO_BYTE(#sxParameter[#piCount].siIndex);
         #sxChaParaMulti.sxData[#piPointer + 4] := WORD_TO_BYTE(SHR(IN := INT_TO_WORD(#sxParameter[#piCount].siIndex), N := 8));

         // Zeiger auf nächsten Parameteradresse setzen
         #piPointer := #piPointer + 6;
       END_FOR; // Auftrags-PARAMETERADRESSE erstellen

       // Auftrags-PARAMETERVALUE erstellen
       FOR #piCount := 1 TO #siParaNo DO

         // Format (BYTE, WORD, DWORD des Parameterwert übergeben
         #sxChaParaMulti.sxData[#piPointer] := #sxParameter[#piCount].syFormat;

         // Number of value
         #sxChaParaMulti.sxData[#piPointer + 1] := B#16#01;

         // Value of parameter in Bytes
         IF (#sxParameter[#piCount].syFormat = B#16#41) OR
           (#sxParameter[#piCount].syFormat = B#16#02) OR (#sxParameter[#piCount].syFormat = B#16#05) THEN

           #sxChaParaMulti.sxData[#piPointer + 2] := WORD_TO_BYTE(DWORD_TO_WORD(DINT_TO_DWORD(REAL_TO_DINT(#sxParameter[#piCount].srValue))));
           #sxChaParaMulti.sxData[#piPointer + 3] := 16#00;  //WORD_TO_BYTE(DWORD_TO_WORD(SHR(IN := DINT_TO_DWORD(REAL_TO_DINT(#sxParameter[#piCount].srValue)), N := 8)));

           // Zeiger auf nächsten Parameteradresse setzen
           #piPointer := #piPointer + 4;

           // Value of parameter in Word
         ELSIF (#sxParameter[#piCount].syFormat = B#16#42) OR
           (#sxParameter[#piCount].syFormat = B#16#03) OR (#sxParameter[#piCount].syFormat = B#16#06) THEN

           #sxChaParaMulti.sxData[#piPointer + 3] := WORD_TO_BYTE(DWORD_TO_WORD(DINT_TO_DWORD(REAL_TO_DINT(#sxParameter[#piCount].srValue))));
           #sxChaParaMulti.sxData[#piPointer + 2] := WORD_TO_BYTE(DWORD_TO_WORD(SHR(IN := DINT_TO_DWORD(REAL_TO_DINT(#sxParameter[#piCount].srValue)), N := 8)));

           // Zeiger auf nächsten Parameteradresse setzen
           #piPointer := #piPointer + 4;

           // Value of parameter in DWord (Double Word ohne Vorzeichen/Double Word mit Vorzeichen)   
         ELSIF (#sxParameter[#piCount].syFormat = B#16#43) OR (#sxParameter[#piCount].syFormat = B#16#04) OR
           (#sxParameter[#piCount].syFormat = B#16#07) THEN

           #sxChaParaMulti.sxData[#piPointer + 5] := WORD_TO_BYTE(DWORD_TO_WORD(DINT_TO_DWORD(#sxParameter[#piCount].sdValue)));
           #sxChaParaMulti.sxData[#piPointer + 4] := WORD_TO_BYTE(DWORD_TO_WORD(SHR(IN := DINT_TO_DWORD(#sxParameter[#piCount].sdValue), N := 8)));
           #sxChaParaMulti.sxData[#piPointer + 3] := WORD_TO_BYTE(DWORD_TO_WORD(SHR(IN := DINT_TO_DWORD(#sxParameter[#piCount].sdValue), N := 16)));
           #sxChaParaMulti.sxData[#piPointer + 2] := WORD_TO_BYTE(DWORD_TO_WORD(SHR(IN := DINT_TO_DWORD(#sxParameter[#piCount].sdValue), N := 24)));

           // Zeiger auf nächsten Parameteradresse setzen
           #piPointer := #piPointer + 6;

           // Value of parameter in DWord (FloatingPoint)   
         ELSIF (#sxParameter[#piCount].syFormat = B#16#08) THEN

           #sxChaParaMulti.sxData[#piPointer + 5] := WORD_TO_BYTE(DWORD_TO_WORD(REAL_TO_DWORD(#sxParameter[#piCount].srValue)));
           #sxChaParaMulti.sxData[#piPointer + 4] := WORD_TO_BYTE(DWORD_TO_WORD(SHR(IN := REAL_TO_DWORD(#sxParameter[#piCount].srValue), N := 8)));
           #sxChaParaMulti.sxData[#piPointer + 3] := WORD_TO_BYTE(DWORD_TO_WORD(SHR(IN := REAL_TO_DWORD(#sxParameter[#piCount].srValue), N := 16)));
           #sxChaParaMulti.sxData[#piPointer + 2] := WORD_TO_BYTE(DWORD_TO_WORD(SHR(IN := REAL_TO_DWORD(#sxParameter[#piCount].srValue), N := 24)));

           // Zeiger auf nächsten Parameteradresse setzen
           #piPointer := #piPointer + 6;
         END_IF;
       END_FOR; // Auftrags-PARAMETERVALUE erstellen 

       // SCHREIBEN AZYKLISCH
       #piLenTele := #siLenHeader + #siLenChaPara;
       #WRREC_1(REQ := True,                                // Startimpuls
                ID := #hardwareId,                         // Diagnoseadresse
                INDEX := 47,                                  // Rahmentyp
                LEN := INT_TO_UINT(#piLenTele),             // maximale Länge
                DONE => #sbWrDone,                           // Schreibauftrag beendet
                BUSY => #sbWrBusy,                           // Slave beschäftigt
                ERROR => #sbWrError,                          // Fehler beim Schreiben
                STATUS => #pdStatus,                           // Status[1] = Error => Status[2] Error Decode + Status[3] Error Code
                RECORD := #sxChaParaMulti);                    // Zeiger auf zu schreibenen Datensatzes

       // Ausgänge setzen
       #sbBusy := #sbWrBusy;
       #sbDone := #sbWrDone;

       // Fehler auswerten
       IF #sbWrError THEN
         // Fehlerstatus aus dem Doppelwort filtern und weitergeben                
         #pwWord1 := DWORD_TO_WORD(SHR(IN := (#pdStatus AND DW#16#FFFF00), N := 8));

         // Fehlerstatus setzen
         #siErrorId := 3;
         #sbError := False;
         #DiagId := #pwWord1;

         //Temporärer Fehler: #pdStatus = 80A7, 80B5, 80C0, 80C1, 80C2, 80C3 oder 80C4 zulassen und nocheinmal versuchen
         IF NOT (#pwWord1 = DW#16#80A7) AND NOT (#pwWord1 = DW#16#80B5) AND NOT (#pwWord1 = DW#16#80C0) AND
           NOT (#pwWord1 = DW#16#80C1) AND NOT (#pwWord1 = DW#16#80C2) AND NOT (#pwWord1 = DW#16#80C3) AND
           NOT (#pwWord1 = DW#16#80C4) THEN

           // Wiederholungsauftrag wieder zurücknehmen
           #sbWrStart2 := False;
           #sbRdStart2 := False;
           #sbWrite := False;

           // Fehler ausgeben 
           #sbError := #sbWrError;

         ELSE
           // Fehlerwiederholauftrag ??                   
           IF #siErrorCount = #siMaxErrCount THEN

             // Wiederholungsauftrag wieder zurücknehmen
             #sbWrStart2 := False;
             #sbRdStart2 := False;
             #sbWrite := False;

             //Fehlerzähler zurücksetzen
             #siErrorCount := 0;

             // Fehler ausgeben 
             #sbError := #sbWrError;

             // nix tun bis Zähler überläuft
           ELSE
             #siErrorCount := #siErrorCount + 1;
           END_IF;
         END_IF;

         // kein Fehler beim SCHEIBEN AZYKLISCH und Auftrag fertig 
       ELSIF NOT #sbWrBusy AND #sbWrDone THEN
         // Fehlerkennung zurücknehmen
         #DiagId := W#16#00;

         // Schreibauftrag fertig melden und Leseantrag anstossen
         #sbWrStart2 := False;
         #sbRdStart2 := True;
       END_IF;
     END_IF; // 2. Teilauftrag "Parameter schreiben bzw. ändern" vorbereiten und abschicken

     // vom 2. Teilauftrag "Parameter schreiben bzw. ändern" die Antwort abwarten und dann auswerten
     IF #sbRdStart2 THEN

       // Ablöschen des Empfangspuffers
       #sxRespParaMulti.sxHeader.syReqRef := B#16#00;
       #sxRespParaMulti.sxHeader.syReqId := B#16#00;
       #sxRespParaMulti.sxHeader.syAxisNo := B#16#00;
       #sxRespParaMulti.sxHeader.syParaNo := B#16#00;

       FOR #piCount := 1 TO #siLenParaMulti DO
         #sxRespParaMulti.sxData[#piCount] := B#16#00;
       END_FOR;

       // LESEN AZYKLISCH
       #piLenTele := #siLenHeader + #siLenParaMulti;
       #RDREC_1(REQ := True,                                // Startimpuls
                ID := #hardwareId,                         // Diagnoseadresse        
                INDEX := 47,                                  // Rahmentyp           
                MLEN := INT_TO_UINT(#piLenTele),             // maximale Länge
                VALID => #pbValidSFB,                         // neuer Datensatz empfangen und gültig   
                BUSY => #sbRdBusy,                           // Slave beschäftigt
                ERROR => #sbRdError,                          // Fehler beim Schreiben
                STATUS => #pdStatus,                           // Status[1] = Error => Status[2] Error Decode + Status[3] Error Code 
                LEN => #piLenSFB,                           // Länge des gelesenen Datensatzes
                RECORD := #sxRespParaMulti);                   // Zeiger auf gelesenen Datensatz

       // Ausgänge setzen
       #sbBusy := #sbRdBusy;
       #sbDone := #pbValidSFB;

       // Fehler auswerten
       IF #sbRdError THEN
         // Fehlerstatus aus dem Doppelwort filtern und weitergeben                
         #pwWord1 := DWORD_TO_WORD(SHR(IN := (#pdStatus AND DW#16#FFFF00), N := 8));

         // Fehlerstatus setzen
         #siErrorId := 3;
         #DiagId := #pwWord1;

         //Temporärer Fehler: #pdStatus = 80A7, 80B5, 80C0, 80C1, 80C2, 80C3 oder 80C4 zulassen und nocheinmal versuchen
         IF NOT (#pwWord1 = DW#16#80A7) AND NOT (#pwWord1 = DW#16#80B5) AND NOT (#pwWord1 = DW#16#80C0) AND
           NOT (#pwWord1 = DW#16#80C1) AND NOT (#pwWord1 = DW#16#80C2) AND NOT (#pwWord1 = DW#16#80C3) AND
           NOT (#pwWord1 = DW#16#80C4) THEN

           // Wiederholungsauftrag wieder zurücknehmen
           #sbWrStart2 := False;
           #sbRdStart2 := False;
           #sbWrite := False;

           // Fehler ausgeben 
           #sbError := #sbRdError;

         ELSE
           // Fehlerwiederholauftrag ??                   
           IF #siErrorCount = #siMaxErrCount THEN

             // Wiederholungsauftrag wieder zurücknehmen
             #sbWrStart2 := False;
             #sbRdStart2 := False;
             #sbWrite := False;

             //Fehlerzähler zurücksetzen
             #siErrorCount := 0;

             // Fehler ausgeben 
             #sbError := #sbRdError;

             // nix tun bis Zähler überläuft
           ELSE
             #siErrorCount := #siErrorCount + 1;
           END_IF;
         END_IF;

         // Fehler : die Auftragsreferenz der Antwort übertimmt nicht mit der Auftragsreferenz der Anfrage überein
       ELSIF NOT (#siReqRef = BYTE_TO_INT(#sxRespParaMulti.sxHeader.syReqRef)) AND NOT #sbRdBusy AND #pbValidSFB THEN
         #siErrorId := 1;
         #sbError := True;
         #sbDone := False;

         // Wiederholungsauftrag wieder zurücknehmen
         #sbWrStart2 := False;
         #sbRdStart2 := False;
         #sbWrite := False;

         // Fehler : falsche Auftragskennung zurück erhalten    
       ELSIF NOT (#sxRespParaMulti.sxHeader.syReqId = B#16#82 OR #sxRespParaMulti.sxHeader.syReqId = B#16#02) AND
         NOT #sbRdBusy AND #pbValidSFB THEN
         #siErrorId := 1;
         #sbError := True;
         #sbDone := False;

         // Wiederholungsauftrag wieder zurücknehmen
         #sbWrStart2 := False;
         #sbRdStart2 := False;
         #sbWrite := False;

         // Fehler : die angeforderte Anzahl Parameter entspricht nicht der übermittelten Anzahl Parameter überein
       ELSIF NOT (#siParaNo = BYTE_TO_INT(#sxRespParaMulti.sxHeader.syParaNo)) AND NOT #sbRdBusy AND #pbValidSFB THEN
         #siErrorId := 1;
         #sbError := True;
         #sbDone := False;

         // Wiederholungsauftrag wieder zurücknehmen
         #sbWrStart2 := False;
         #sbRdStart2 := False;
         #sbWrite := False;

         // Fehler : die Achse entspricht nicht der übergebenen Achse
       ELSIF NOT (#syAxisNo = #sxRespParaMulti.sxHeader.syAxisNo) AND NOT #sbRdBusy AND #pbValidSFB THEN
         #siErrorId := 1;
         #sbError := True;
         #sbDone := False;

         // Wiederholungsauftrag wieder zurücknehmen
         #sbWrStart2 := False;
         #sbRdStart2 := False;
         #sbWrite := False;

         // kein Fehler beim LESEN AZYKLISCH und Auftrag fertig 
       ELSIF NOT #sbRdBusy AND #pbValidSFB THEN

         // 2. Teilauftrag "Parameter schreiben bzw. ändern" negative Rückmeldung erhalten 
         IF #sxRespParaMulti.sxHeader.syReqId = B#16#82 THEN

           // die angefragten Parameter auswerten und im Puffer abspeichern
           #piPointer := 1;
           #swParaError := 16#0;

           FOR #piCount := 1 TO #siParaNo DO

             // Format des Parameters auswerten, bei Format = Error Fehler auswerten 
             IF (BYTE_TO_INT(#sxRespParaMulti.sxData[#piPointer]) = 68) THEN

               // Fehlerwert ermitteln und abspeichern 
               // Format = Word, zwei Bytes zu übermitteltem Parameterwert zusammenfassen
               #pwWordHigh := SHL(IN := BYTE_TO_WORD(#sxRespParaMulti.sxData[#piPointer + 2]), N := 8);
               #pwWordLow := BYTE_TO_WORD(#sxRespParaMulti.sxData[#piPointer + 3]);
               #pwWord1 := #pwWordHigh XOR #pwWordLow;

               #sbError := True;

               // ermittelte Fehlernummer im Puffer zurücksetzen
               #sxParameter[#piCount].swErrorNo := W#16#00;

               #sxParameter[#piCount].swErrorNo := #pwWord1;

               // Die Fehlerhaftigkeit des erkannten Parameter in der Fehlernummer eintragen   
               IF #piCount = 1 THEN
                 #swParaError := #swParaError OR W#16#01;
               ELSIF #piCount = 2 THEN
                 #swParaError := #swParaError OR W#16#02;
               ELSIF #piCount = 3 THEN
                 #swParaError := #swParaError OR W#16#04;
               ELSIF #piCount = 4 THEN
                 #swParaError := #swParaError OR W#16#08;
               ELSIF #piCount = 5 THEN
                 #swParaError := #swParaError OR W#16#10;
               ELSIF #piCount = 6 THEN
                 #swParaError := #swParaError OR W#16#20;
               ELSIF #piCount = 7 THEN
                 #swParaError := #swParaError OR W#16#40;
               ELSIF #piCount = 8 THEN
                 #swParaError := #swParaError OR W#16#80;
               ELSIF #piCount = 9 THEN
                 #swParaError := #swParaError OR W#16#100;
               ELSIF #piCount = 10 THEN
                 #swParaError := #swParaError OR W#16#200;
               ELSIF #piCount = 11 THEN
                 #swParaError := #swParaError OR W#16#400;
               ELSIF #piCount = 12 THEN
                 #swParaError := #swParaError OR W#16#800;
               ELSIF #piCount = 13 THEN
                 #swParaError := #swParaError OR W#16#1000;
               ELSIF #piCount = 14 THEN
                 #swParaError := #swParaError OR W#16#2000;
               ELSIF #piCount = 15 THEN
                 #swParaError := #swParaError OR W#16#4000;
               ELSIF #piCount = #siParaNo THEN
                 #swParaError := #swParaError OR W#16#8000;
               END_IF;

               // Zeiger auf nächsten Parametersatz setzen
               #piPointer := #piPointer + 6;
             ELSE
               // Zeiger auf nächsten Parametersatz setzen
               #piPointer := #piPointer + 2;

               // Die Fehlerhaftigkeit des erkannten Parameter in der Fehlernummer löschen   
               IF #piCount = 1 THEN
                 #swParaError := #swParaError AND W#16#FFFE;
               ELSIF #piCount = 2 THEN
                 #swParaError := #swParaError AND W#16#FFFD;
               ELSIF #piCount = 3 THEN
                 #swParaError := #swParaError AND W#16#FFFB;
               ELSIF #piCount = 4 THEN
                 #swParaError := #swParaError AND W#16#FFF7;
               ELSIF #piCount = 5 THEN
                 #swParaError := #swParaError AND W#16#FFEF;
               ELSIF #piCount = 6 THEN
                 #swParaError := #swParaError AND W#16#FFDF;
               ELSIF #piCount = 7 THEN
                 #swParaError := #swParaError AND W#16#FFBF;
               ELSIF #piCount = 8 THEN
                 #swParaError := #swParaError AND W#16#FF7F;
               ELSIF #piCount = 9 THEN
                 #swParaError := #swParaError AND W#16#FEFF;
               ELSIF #piCount = 10 THEN
                 #swParaError := #swParaError AND W#16#FDFF;
               ELSIF #piCount = 11 THEN
                 #swParaError := #swParaError AND W#16#FBFF;
               ELSIF #piCount = 12 THEN
                 #swParaError := #swParaError AND W#16#F7FF;
               ELSIF #piCount = 13 THEN
                 #swParaError := #swParaError AND W#16#EFFF;
               ELSIF #piCount = 14 THEN
                 #swParaError := #swParaError AND W#16#DFFF;
               ELSIF #piCount = 15 THEN
                 #swParaError := #swParaError AND W#16#BFFF;
               ELSIF #piCount = #siParaNo THEN
                 #swParaError := #swParaError AND W#16#7FFF;
               END_IF;

               // ermittelte Fehlernummer im Puffer zurücksetzen
               #sxParameter[#piCount].swErrorNo := W#16#00;
             END_IF;
           END_FOR; // die angefragten Parameter auswerten und im Puffer abspeichern
         END_IF; // 2. Teilauftrag "Parameter schreiben bzw. ändern" negative Rückmeldung erhalten

         // Fehlerkennung zurücknehmen
         IF (#siErrorId = 3) OR (#siErrorId = 1) THEN
           #siErrorId := 0;
           #sbError := False;
         END_IF;

         #DiagId := W#16#00;

         // 2. Teilauftrag "Parameter schreiben bzw. ändern" ist abgeschlossen
         #sbRdStart2 := False;
         #sbWrite := False;

       END_IF; // kein Fehler beim LESEN AZYKLISCH und Auftrag fertig 
     END_IF; // vom 2. Teilauftrag "Parameter schreiben bzw. ändern" die Antwort abwarten und dann auswerten 
   END_IF; // Auftrag "Parameter schreiben" wurde ausgelöst

   #pdDWordHigh := SHL(IN := INT_TO_DWORD(#siErrorId), N := 16);
   #pdDWordLow := WORD_TO_DWORD(#swParaError);

   // ermittelter Parameterwert eintragen (Word)
   #ErrorId := #pdDWordHigh XOR #pdDWordLow;

   // Initialisierung von Ausgängen
   #Busy := #sbBusy;
   #Error := #sbError;
   // Änderung wegen verhalten von Ready  
   #Done := #sbDone;
   // Prüfen, ob Auftrag abgeschlossen ist
   IF ((#Error OR #Done) AND NOT #sbReady) THEN
     #Ready := True;
     #sbReady := True;
   ELSE
     #Ready := False;
   END_IF;
END_FUNCTION_BLOCK

FUNCTION "LGF_BitsToWord" : Word   // FC10044, SCL
{ S7_Optimized_Access := 'TRUE' }
VERSION : 0.1
   VAR_INPUT
      bit0 : Bool;
      bit1 : Bool;
      bit2 : Bool;
      bit3 : Bool;
      bit4 : Bool;
      bit5 : Bool;
      bit6 : Bool;
      bit7 : Bool;
      bit8 : Bool;
      bit9 : Bool;
      bit10 : Bool;
      bit11 : Bool;
      bit12 : Bool;
      bit13 : Bool;
      bit14 : Bool;
      bit15 : Bool;
   END_VAR
BEGIN
   //=============================================================================
   // SIEMENS AG
   // (c)Copyright 2017
   //-----------------------------------------------------------------------------
   // Library:       LGF(Library General Functions)
   // Tested with:   CPU1212C DC/DC/DC FW:V4.2
   // Engineering:   TIA Portal V14 Update 1
   // Restrictions:  -
   // Requirements:  PLC (S7-1200 / S7-1500)
   // Functionality: This function converts 16 bits to a word
   //-----------------------------------------------------------------------------
   // Change log table:
   // Version  Date        In charge / Changes applied
   // 01.00.00 09.02.2017  Siemens Industry Online Support
   //                      First released version
   //=============================================================================

   #LGF_BitsToWord.%X0 := #bit0;
   #LGF_BitsToWord.%X1 := #bit1;
   #LGF_BitsToWord.%X2 := #bit2;
   #LGF_BitsToWord.%X3 := #bit3;
   #LGF_BitsToWord.%X4 := #bit4;
   #LGF_BitsToWord.%X5 := #bit5;
   #LGF_BitsToWord.%X6 := #bit6;
   #LGF_BitsToWord.%X7 := #bit7;
   #LGF_BitsToWord.%X8 := #bit8;
   #LGF_BitsToWord.%X9 := #bit9;
   #LGF_BitsToWord.%X10 := #bit10;
   #LGF_BitsToWord.%X11 := #bit11;
   #LGF_BitsToWord.%X12 := #bit12;
   #LGF_BitsToWord.%X13 := #bit13;
   #LGF_BitsToWord.%X14 := #bit14;
   #LGF_BitsToWord.%X15 := #bit15;
END_FUNCTION

// folder: FB/Controle Automático

FUNCTION_BLOCK "Controle_Automatico"   // FB5, FBD
TITLE = Controle Automático
{ S7_Optimized_Access := 'TRUE' }
VERSION : 0.1
// Maycon Lutz
// 17/07/20
// Controle automático de bateladas fábrica de ração.
   VAR_INPUT
      inPeso_Atual_Silo_Produto_Acabado : Real;
      inPeso_Atual_Balanca_Dosagem : Real;
      inNivel_Inferior_Pre_Mistura : Bool;
      inNivel_Inferior_Pos_Mistura : Bool;
      inNivel_Superior_Silo_Produto_Acabado : Bool;
      inConfiguracoes_Maquinas : Struct
         Maximo_Silo_Produto_Acabado : Real;
         Maximo_Silo_1_Materia_Prima : Real;
         Maximo_Silo_2_Materia_Prima : Real;
         Maximo_Balanca : Real;
         Maximo_PreMisturador : Real;
         Maximo_PosMisturador : Real;
      END_STRUCT;
      inConfiguracoes_Registro_26 : Struct
         Abertura_Maxima_Silo_1 : Real;   // Percentual de abertura máximo do registro 26 Silo 1
         Inicio_Reducao_Silo_1 : Real;   // Percentual do inicio da redução do registro 26 Silo 1
         Fechamento_Antecipado_Silo_1 : Real;
         Abertura_Maxima_Silo_2 : Real;   // Percentual de abertura máximo do registro 26 Silo 2
         Inicio_Reducao_Silo_2 : Real;   // Percentual do inicio da redução do registro 26 Silo 2
         Fechamento_Antecipado_Silo_2 : Real;
      END_STRUCT;
   END_VAR
   VAR_OUTPUT
      outPosicao_Atuador_Silo_1 : Real;
      outPosicao_Atuador_Silo_2 : Real;
      outSolicita_Dosagem_Complemento_Pre : Bool;
      outSolicita_Dosagem_Complemento_Pos : Bool;
   END_VAR
   VAR_IN_OUT
      inOutControle : Struct
         Dosagem_Materia_Prima : Struct
            Ligar : Bool;   // Solicita ligar Dosagem
            Ligado : Bool;   // Dosagem Ligada
            Liberado_Nova_Dosagem : Bool;   // Liberado dosagem de nova batelada
            Finalizado_Dosagem : Bool;   // finalizado dosagem da batelada solicitada
            Balanca_Vazia : Bool;   // Solicita balança vazia
            Habilita_Setar_Balanca_Vazia : Bool;   // habilita solicitar balança vazia
            Reserva : Bool;
            Reserva_1 : Bool;
            Passo_Atual : Int;   // Passo Atual da dosagem
            Dosagem_Materia_Prima_Silo_1 : Real;   // Valor em Kg da dosagem de materia prima do silo 1 solicitada
            Dosagem_Materia_Prima_Silo_2 : Real;   // Valor em Kg da dosagem de materia prima do silo 2 solicitada
            Dosado_Materia_Prima_Silo_1 : Real;   // Valor dosado do silo 1 na balança
            Dosado_Materia_Prima_Silo_2 : Real;   // Valor dosado do silo 2 na balança
            Complemento_Pre : Struct   // Complementos dosados manualmente na balança
               Quantidade_Itens : Int;   // Quantidade de complementos na receita
               Item_Atual : Int;   // Em qual item da receita esta no momento
               Quantidade_Dosada_Item_Atual : Real;   // Quantidade dosada do item atual, valor disponível após finalizado dosagem
               Habilitado_Inicio_Dosagem : Bool;   // Habilita o inicio da dosagem manual
               Botao_Inicio_Fim_Dosagem_IHM : Bool;   // Bit para iniciar ou finalizar dosagem pela IHM
               Item_Atual_Iniciado_Dosagem : Bool;   // Se iniciou a dosagem do item atual
               Item_Atual_Finalizado_Dosagem : Bool;   // Se finalizou a dosagem do item atual
               Finalizado_Dosagem_Complementos : Bool;   // Se finalizou a dosagem de todos os complementos
               Reserva : Bool;
               Reserva_1 : Bool;
               Reserva_2 : Bool;
            END_STRUCT;
         END_STRUCT;
         Transporte_Para_Pre_Mistura : Struct
            Ligar : Bool;   // Solicita ligar transporte
            Ligado : Bool;   // Transporte ligado
            Liberado_Iniciar_Transporte : Bool;   // liberado iniciar transporte
            Reserva : Bool;
            Reserva_1 : Bool;
            Reserva_2 : Bool;
            Reserva_3 : Bool;
            Reserva_4 : Bool;
         END_STRUCT;
         Pre_Mistura : Struct
            Ligar : Bool;   // Solicita ligar pré mistura
            Ligado : Bool;   // Pré mistura ligado
            Liberado_Nova_Batelada : Bool;   // Liberado mistura de nova batelada
            Recebendo_Produto : Bool;   // Esta recebendo produto
            Iniciado_Mistura : Bool;   // Iniciado a mistura
            Finalizado_Mistura : Bool;   // Finalizado mistura
            Reserva : Bool;
            Reserva_1 : Bool;
            Tempo_SP : DInt;   // Tempo em segundos de mistura
            Tempo_Restante : DInt;   // Tempo em segundos restante
         END_STRUCT;
         Moagem_Pos_Mistura : Struct
            Ligar : Bool;   // Solicita ligar moagem
            Ligado : Bool;   // Moagem ligado
            Liberado_Nova_Moagem : Bool;   // Liberado moagem de nova batelada
            Finalizou_Moagem : Bool;   // Finalizou Moagem
            Reserva : Bool;
            Reserva_1 : Bool;
            Reserva_2 : Bool;
            Reserva_3 : Bool;
         END_STRUCT;
         Pos_Mistura : Struct
            Ligar : Bool;   // Solicita ligar pós mistura
            Ligado : Bool;   // pós mistura ligado
            Liberado_Nova_Batelada : Bool;   // liberado mistura de nova batelada
            Recebendo_Produto : Bool;   // Esta recebendo produto
            Iniciado_Mistura : Bool;   // Iniciado a mistura
            Finalizado_Mistura : Bool;   // Finalizado mistura
            Reserva : Bool;
            Reserva_1 : Bool;
            Tempo_SP : DInt;   // Tempo em segundos de mistura
            Tempo_Restante : DInt;   // Tempo em segundos restante
            Complemento_Pos : Struct   // Complementos dosados manualmente
               Quantidade_Itens : Int;   // Quantidade de complementos na receita
               Item_Atual : Int;   // Em qual item da receita esta no momento
               Quantidade_Dosada_Item_Atual : Real;   // Quantidade dosada do item atual, valor disponível após finalizado dosagem
               Habilitado_Inicio_Dosagem : Bool;   // Habilita o inicio da dosagem manual
               Botao_Inicio_Fim_Dosagem_IHM : Bool;   // Bit para iniciar ou finalizar dosagem pela IHM
               Item_Atual_Iniciado_Dosagem : Bool;   // Se iniciou a dosagem do item atual
               Item_Atual_Finalizado_Dosagem : Bool;   // Se finalizou a dosagem do item atual
               Finalizado_Dosagem_Complementos : Bool;   // Se finalizou a dosagem de todos os complementos
               Reserva : Bool;
               Reserva_1 : Bool;
               Reserva_2 : Bool;
            END_STRUCT;
         END_STRUCT;
         Transporte_Produto_Acabado : Struct
            Ligar : Bool;   // Solicita ligar transporte para produto acabado
            Ligado : Bool;   // Transporte para produto acabado ligado
            Liberado_Iniciar_Transporte : Bool;   // Liberado transporte nova batelada para produto acabado
            Reserva : Bool;
            Reserva_1 : Bool;
            Reserva_2 : Bool;
            Reserva_3 : Bool;
            Reserva_4 : Bool;
         END_STRUCT;
      END_STRUCT;
   END_VAR
   VAR
      Valor_Inicio_Dosagem_Silo1 : Real;
      Valor_Inicio_Dosagem_Silo2 : Real;
      Controle_Descarga_Atuador_Linear_Silo1 : "Controle_Descarga_Atuador_Linear";
      Controle_Descarga_Atuador_Linear_Silo2 : "Controle_Descarga_Atuador_Linear";
      Controle_Dosagem_Complementos_Pre : "Controle_Dosagem_Complementos";
      Controle_Dosagem_Complementos_Pos : "Controle_Dosagem_Complementos";
      Temporizador_Pre_Mistura : TON_TIME;
      Temporizador_Pos_Mistura : TON_TIME;
      Finalizado_Transporte_Pre_Mistura : Bool;   // Finalizado o transporte da balança para a pré mistura
      Temporizador_Finalizado_Transporte_Pre_Mistura : TON_TIME;
      Moagem_Sem_Carga : Bool;
      Tempo_Moagem_Sem_Carga : TON_TIME;
      Finalizado_Transporte_Pos_Mistura : Bool;
      Temporizador_Finalizado_Transporte_Pos_Mistura : TON_TIME;
      Elevador_62_Sem_Carga : Bool;
      Tempo_Transporte_Para_Produto_Acabado : TON_TIME;
   END_VAR
BEGIN

REGION Network 1 (SCL): Dosagem Matéria Prima
   //Passo 20 - Dosa na balança o que foi solicitado para dosar a partir do silo 1
   //Passo 21 - Dosa na balança o que foi solicitado para dosar a partir do silo 2
   //Passo 22 - Dosagem manual dos complementos na balança

   //Quando solicitar ligar e esta liberado
   //seta a balança para não vazia
   //seta como ligado a dosagem de materia prima
   //reseta o liberado para nova dosagem
   //inicia no passo 20
   IF #inOutControle.Dosagem_Materia_Prima.Ligar AND
      #inOutControle.Dosagem_Materia_Prima.Liberado_Nova_Dosagem THEN
      #inOutControle.Dosagem_Materia_Prima.Balanca_Vazia := false;
      #inOutControle.Dosagem_Materia_Prima.Ligado := true;
      #inOutControle.Dosagem_Materia_Prima.Liberado_Nova_Dosagem := false;
      #inOutControle.Dosagem_Materia_Prima.Passo_Atual := 20;

   END_IF;

   //------------------------------------------------------------------------------------------------------------
   //Dosagem Matéria Prima - Verifica se tem dosagem do silo 1, se tem realiza a dosagem (Liga atuador linear).
   IF #inOutControle.Dosagem_Materia_Prima.Passo_Atual = 20 THEN

       IF #inOutControle.Dosagem_Materia_Prima.Dosagem_Materia_Prima_Silo_1 = 0 THEN
           #inOutControle.Dosagem_Materia_Prima.Passo_Atual := 21;
       ELSE

           #Controle_Descarga_Atuador_Linear_Silo1.inDosar := true;

           IF #Controle_Descarga_Atuador_Linear_Silo1.outDosagem_Finalizada THEN
           #inOutControle.Dosagem_Materia_Prima.Passo_Atual := 21;
       END_IF;

       END_IF;

   ELSE

       #Controle_Descarga_Atuador_Linear_Silo1.inDosar := false;

   END_IF;

   //Controle de dosagem Silo 1 de matéria prima
   #Controle_Descarga_Atuador_Linear_Silo1(inValor_Dosar := #inOutControle.Dosagem_Materia_Prima.Dosagem_Materia_Prima_Silo_1,
                                      inValor_Atual_Balanca := #inPeso_Atual_Balanca_Dosagem,
                                      inAbertura_Maxima_Atuador := #inConfiguracoes_Registro_26.Abertura_Maxima_Silo_1,
                                      inInicio_Reducao := #inConfiguracoes_Registro_26.Inicio_Reducao_Silo_1,
                                      inFechamento_Antecipado := #inConfiguracoes_Registro_26.Fechamento_Antecipado_Silo_1,
                                      outPosicao_Atuador => #outPosicao_Atuador_Silo_1,
                                      outValor_Dosado_Ultima_Dosagem=>#inOutControle.Dosagem_Materia_Prima.Dosado_Materia_Prima_Silo_1);

   //------------------------------------------------------------------------------------------------------------
   //Passo 2.1 - Verifica se tem dosagem do silo 2, se tem realiza a dosagem (Liga atuador linear).
   IF #inOutControle.Dosagem_Materia_Prima.Passo_Atual = 21 THEN

       IF #inOutControle.Dosagem_Materia_Prima.Dosagem_Materia_Prima_Silo_2 = 0 THEN
           #inOutControle.Dosagem_Materia_Prima.Passo_Atual := 22;
       ELSE

           #Controle_Descarga_Atuador_Linear_Silo2.inDosar := true;

           IF #Controle_Descarga_Atuador_Linear_Silo2.outDosagem_Finalizada THEN
               #inOutControle.Dosagem_Materia_Prima.Passo_Atual := 22;
           END_IF;

       END_IF;

   ELSE

       #Controle_Descarga_Atuador_Linear_Silo2.inDosar := false;

   END_IF;

   //Controle de dosagem Silo 1 de matéria prima
   #Controle_Descarga_Atuador_Linear_Silo2(inValor_Dosar := #inOutControle.Dosagem_Materia_Prima.Dosagem_Materia_Prima_Silo_2,
                                      inValor_Atual_Balanca := #inPeso_Atual_Balanca_Dosagem,
                                      inAbertura_Maxima_Atuador := #inConfiguracoes_Registro_26.Abertura_Maxima_Silo_2,
                                      inInicio_Reducao := #inConfiguracoes_Registro_26.Inicio_Reducao_Silo_2,
                                      inFechamento_Antecipado := #inConfiguracoes_Registro_26.Fechamento_Antecipado_Silo_2,
                                      outPosicao_Atuador => #outPosicao_Atuador_Silo_2,
                                      outValor_Dosado_Ultima_Dosagem => #inOutControle.Dosagem_Materia_Prima.Dosado_Materia_Prima_Silo_2);

   //------------------------------------------------------------------------------------------------------------
   //Passo 2.2 - Verifica se tem dosagem de complementos, se tem solicita a dosagem dos complementos da receita.

   #Controle_Dosagem_Complementos_Pre(inEnable:= #inOutControle.Dosagem_Materia_Prima.Passo_Atual = 22,
                                   inBotao_Externo:="BT_27_DOSAGEM_MANUAL",
                                   inValor_Atual_Balanca:= #inPeso_Atual_Balanca_Dosagem,
                                   outLedBotao_Externo=>"LIGA_LED_BT_27_DOSAGEM_MANUAL",
                                   Controle:=#inOutControle.Dosagem_Materia_Prima.Complemento_Pre);

   //Verifica se foi finalizado a dosagem de complementos, se sim, finaliza a dosagem da matéria prima.
   IF #inOutControle.Dosagem_Materia_Prima.Complemento_Pre.Finalizado_Dosagem_Complementos AND
       #inOutControle.Dosagem_Materia_Prima.Passo_Atual = 22
   THEN
       #inOutControle.Dosagem_Materia_Prima.Passo_Atual := 0;
       #inOutControle.Dosagem_Materia_Prima.Finalizado_Dosagem := true;
   END_IF;

   //Habilita setar balança vazia para habilitar próxima dosagem
   IF #inPeso_Atual_Balanca_Dosagem < 20 AND
       #inOutControle.Dosagem_Materia_Prima.Finalizado_Dosagem = true AND
       #inOutControle.Dosagem_Materia_Prima.Ligado
   THEN

       #inOutControle.Dosagem_Materia_Prima.Habilita_Setar_Balanca_Vazia := true;

   ELSE

       #inOutControle.Dosagem_Materia_Prima.Habilita_Setar_Balanca_Vazia := false;
   END_IF;

   //Balança Vazia
   IF #inOutControle.Dosagem_Materia_Prima.Balanca_Vazia THEN
       #inOutControle.Dosagem_Materia_Prima.Ligar := false;
       #inOutControle.Dosagem_Materia_Prima.Ligado := false;
       #inOutControle.Dosagem_Materia_Prima.Liberado_Nova_Dosagem := true;
       #inOutControle.Dosagem_Materia_Prima.Finalizado_Dosagem := false;
       #inOutControle.Dosagem_Materia_Prima.Dosado_Materia_Prima_Silo_1 := 0;
       #inOutControle.Dosagem_Materia_Prima.Dosado_Materia_Prima_Silo_2 := 0;
   END_IF;

   //Desliga Dosagem e reinicia
   IF NOT #inOutControle.Dosagem_Materia_Prima.Ligar AND NOT #inOutControle.Dosagem_Materia_Prima.Finalizado_Dosagem THEN
       #inOutControle.Dosagem_Materia_Prima.Ligado := false;
       #inOutControle.Dosagem_Materia_Prima.Liberado_Nova_Dosagem := true;
       #inOutControle.Dosagem_Materia_Prima.Passo_Atual := 0;

   END_IF;
END_REGION

REGION Network 2 (SCL): Transporte Para Pré Mistura
   //Liberação Transporte
   ///Verifica se esta finalizado a dosagem e Liberado para transporte da balança para Pré-Mistura
   IF #inOutControle.Dosagem_Materia_Prima.Finalizado_Dosagem AND //Finalizado uma dosagem e esta pronto para transporte
       #inOutControle.Pre_Mistura.Liberado_Nova_Batelada //Pré Mistura, liberado para receber uma nova batelada

   THEN
       #inOutControle.Transporte_Para_Pre_Mistura.Liberado_Iniciar_Transporte := true;

   ELSE
       #inOutControle.Transporte_Para_Pre_Mistura.Liberado_Iniciar_Transporte := false;

   END_IF;


   //Liga transporte para pré mistura
   IF #inOutControle.Dosagem_Materia_Prima.Finalizado_Dosagem AND
       #inOutControle.Transporte_Para_Pre_Mistura.Liberado_Iniciar_Transporte AND
       #inOutControle.Pre_Mistura.Ligado
   THEN
       #inOutControle.Transporte_Para_Pre_Mistura.Ligar := true;

   END_IF;

   //Desliga transporte para pré mistura

   #Temporizador_Finalizado_Transporte_Pre_Mistura(IN := #Finalizado_Transporte_Pre_Mistura,
                                                   PT := t#10s);

   IF #Temporizador_Finalizado_Transporte_Pre_Mistura.Q THEN
       #inOutControle.Transporte_Para_Pre_Mistura.Ligar := false;

   END_IF;


   //Transporte ligado
   IF #inOutControle.Transporte_Para_Pre_Mistura.Ligar = true AND
       "DB_Controle_Equip"."29".ligado AND
       "DB_Controle_Equip"."30".ligado
   THEN
       #inOutControle.Transporte_Para_Pre_Mistura.Ligado := true;

   ELSE
       #inOutControle.Transporte_Para_Pre_Mistura.Ligado := false;
   END_IF;
END_REGION

REGION Network 3 (SCL): Pré-Mistura
   //Ligar pré mistura
   IF #inOutControle.Dosagem_Materia_Prima.Finalizado_Dosagem //Finalizou uma dosagem
   THEN
       #inOutControle.Pre_Mistura.Ligar := true;
   ELSIF NOT #inNivel_Inferior_Pre_Mistura THEN
       #inOutControle.Pre_Mistura.Ligar := false;
   END_IF;


   //Liberado Nova Batelada
   IF NOT #inNivel_Inferior_Pre_Mistura AND
       #inOutControle.Moagem_Pos_Mistura.Liberado_Nova_Moagem //Verifica a moagem pois, os bits para finalizar a moagem são moagem vazio e nível inferior da pré mistura.
       //caso não verificassemos o liberado da nova moagem, poderia ocorrer da moagem não parar entre uma batelada e outra.
   THEN

       #inOutControle.Pre_Mistura.Liberado_Nova_Batelada := true;
       #Finalizado_Transporte_Pre_Mistura := false;

   ELSE
       #inOutControle.Pre_Mistura.Liberado_Nova_Batelada := false;


   END_IF;

   //Verifica se esta ligado
   IF #inOutControle.Pre_Mistura.Ligar AND
       "DB_Controle_Equip"."42".ligado THEN
       #inOutControle.Pre_Mistura.Ligado := true;
   ELSE
       #inOutControle.Pre_Mistura.Ligado := false;
   END_IF;


   //Recebendo Produto
   IF #inOutControle.Pre_Mistura.Ligado AND //Esta ligado a mistura
       #inOutControle.Transporte_Para_Pre_Mistura.Ligado //Esta ligado o transporte para pré mistura
   THEN

       #inOutControle.Pre_Mistura.Recebendo_Produto := true;
   ELSE
       #inOutControle.Pre_Mistura.Recebendo_Produto := false;
   END_IF;


   //Finalizado transporte da balança para pré mistura
   IF #inOutControle.Dosagem_Materia_Prima.Balanca_Vazia AND
       #inOutControle.Pre_Mistura.Ligado
   THEN
       #Finalizado_Transporte_Pre_Mistura := true;
   END_IF;

   //Iniciado Mistura
   IF NOT #inOutControle.Pre_Mistura.Recebendo_Produto AND //Não esta mais recebendo produto
       #inOutControle.Pre_Mistura.Ligado AND //Esta ligado a mistura
       #Finalizado_Transporte_Pre_Mistura
   THEN
       #inOutControle.Pre_Mistura.Iniciado_Mistura := true;
   END_IF;

   //Temporiza o tempo de pré mistura, após ter finalizado todo o transporte da balanaça para pré mistura
   #Temporizador_Pre_Mistura(IN := #inOutControle.Pre_Mistura.Iniciado_Mistura,
                             PT := #inOutControle.Pre_Mistura.Tempo_SP);

   //calcula tempo restante de pré mistura
   #inOutControle.Pre_Mistura.Tempo_Restante := #inOutControle.Pre_Mistura.Tempo_SP - TIME_TO_DINT(#Temporizador_Pre_Mistura.ET);


   //Finalizado Mistura
   IF #Temporizador_Pre_Mistura.Q THEN

       #inOutControle.Pre_Mistura.Finalizado_Mistura := true;
       #inOutControle.Pre_Mistura.Iniciado_Mistura := false;
   ELSE
       #inOutControle.Pre_Mistura.Finalizado_Mistura := false;
   END_IF;
END_REGION

REGION Network 4 (SCL): Moagem e Pós Mistura
   //Liberado Nova Batelada
   IF #inOutControle.Moagem_Pos_Mistura.Finalizou_Moagem OR
       #inOutControle.Pos_Mistura.Liberado_Nova_Batelada
   THEN

       #inOutControle.Moagem_Pos_Mistura.Liberado_Nova_Moagem := true;

   ELSE
       #inOutControle.Moagem_Pos_Mistura.Liberado_Nova_Moagem := false;

   END_IF;


   //Liga Moagem
   IF (#inOutControle.Pre_Mistura.Finalizado_Mistura OR
       (#inOutControle.Moagem_Pos_Mistura.Ligado AND
       NOT #inOutControle.Moagem_Pos_Mistura.Finalizou_Moagem)) AND
       #inOutControle.Pos_Mistura.Ligado

   THEN
       #inOutControle.Moagem_Pos_Mistura.Ligar := true;
       #inOutControle.Moagem_Pos_Mistura.Finalizou_Moagem := false;
   ELSE
       #inOutControle.Moagem_Pos_Mistura.Ligar := false;
   END_IF;



   //Verifica se esta ligado
   IF #inOutControle.Moagem_Pos_Mistura.Ligar AND
       "DB_Controle_Equip"."43".ligado AND
       "DB_Controle_Equip"."44".ligado AND
       "DB_Controle_Equip"."45".ligado AND
       "DB_Controle_Equip"."46".ligado AND
       "DB_Controle_Equip"."48".ligado
   THEN
       #inOutControle.Moagem_Pos_Mistura.Ligado := true;
   ELSE
       #inOutControle.Moagem_Pos_Mistura.Ligado := false;
   END_IF;

   //Moagem sem carga
   IF "DB_Controle_Equip"."44".Corrente_Atual < "DB_Controle_Equip"."44".SP_Corrente_Motor_Vazio AND
       "DB_Controle_Equip"."44".ligado
   THEN
       #Moagem_Sem_Carga := true;
   ELSE
       #Moagem_Sem_Carga := false;
   END_IF;

   #Tempo_Moagem_Sem_Carga(IN := #Moagem_Sem_Carga,
                           PT := t#10s);


   //Finaliza Moagem
   IF #Tempo_Moagem_Sem_Carga.Q AND
       NOT #inNivel_Inferior_Pre_Mistura AND
       #inOutControle.Moagem_Pos_Mistura.Ligado
   THEN
       #inOutControle.Moagem_Pos_Mistura.Finalizou_Moagem := true;
   END_IF;
END_REGION

REGION Network 5 (SCL): Pós mistura
   //Ligar pré mistura
   IF #inOutControle.Moagem_Pos_Mistura.Finalizou_Moagem OR //Finalizou moagem
       #inOutControle.Pre_Mistura.Finalizado_Mistura OR //pré mistura ficar pronta, tem que ligar pós mistura antes, pois a pós mistura que libera o Moinho
       #inOutControle.Moagem_Pos_Mistura.Ligado //Moagem ligado
   THEN
       #inOutControle.Pos_Mistura.Ligar := true;
   ELSIF NOT #inNivel_Inferior_Pos_Mistura THEN
       #inOutControle.Pos_Mistura.Ligar := false;
   END_IF;

   //Liberado Nova Batelada
   IF NOT #inNivel_Inferior_Pos_Mistura THEN

       #inOutControle.Pos_Mistura.Liberado_Nova_Batelada := true;

   ELSE
       #inOutControle.Pos_Mistura.Liberado_Nova_Batelada := false;

   END_IF;

   //Verifica se esta ligado
   IF #inOutControle.Pos_Mistura.Ligar AND
       "DB_Controle_Equip"."48".ligado
   THEN
       #inOutControle.Pos_Mistura.Ligado := true;
   ELSE
       #inOutControle.Pos_Mistura.Ligado := false;
   END_IF;


   //Recebendo Produto
   IF #inOutControle.Pos_Mistura.Ligado AND //Esta ligado a mistura
       #inOutControle.Moagem_Pos_Mistura.Ligado //Esta ligado a moagem para pós mistura
   THEN

       #inOutControle.Pos_Mistura.Recebendo_Produto := true;
   ELSE
       #inOutControle.Pos_Mistura.Recebendo_Produto := false;
   END_IF;

   //Finalizado transporte do moinho para pós mistura
   IF #inOutControle.Moagem_Pos_Mistura.Finalizou_Moagem AND
       #inOutControle.Pos_Mistura.Ligado
   THEN
       #Finalizado_Transporte_Pos_Mistura := true;
   END_IF;

   //Verifica se tem dosagem de complementos POS, se tem solicita a dosagem dos complementos da receita.
   #Controle_Dosagem_Complementos_Pos(inEnable := #Finalizado_Transporte_Pos_Mistura,
                                      inValor_Atual_Balanca := #inPeso_Atual_Balanca_Dosagem,
                                      Controle := #inOutControle.Pos_Mistura.Complemento_Pos);

   //Iniciado Mistura
   IF NOT #inOutControle.Pos_Mistura.Recebendo_Produto AND //Não esta mais recebendo produto
       #inOutControle.Pos_Mistura.Ligado AND //Esta ligado a mistura
       #Finalizado_Transporte_Pos_Mistura AND //Finalizado transporte 
       #inOutControle.Pos_Mistura.Complemento_Pos.Finalizado_Dosagem_Complementos //Finalizou dosagem de complementos se tinha complementos
   THEN
       #inOutControle.Pos_Mistura.Iniciado_Mistura := true;
   END_IF;

   //Temporiza o tempo de pré mistura, após ter finalizado todo o transporte da balanaça para pré mistura
   #Temporizador_Pos_Mistura(IN := #inOutControle.Pos_Mistura.Iniciado_Mistura,
                             PT := #inOutControle.Pos_Mistura.Tempo_SP);

   //calcula tempo restante de pré mistura
   #inOutControle.Pos_Mistura.Tempo_Restante := #inOutControle.Pos_Mistura.Tempo_SP - TIME_TO_DINT(#Temporizador_Pos_Mistura.ET);


   //Finalizado Mistura
   IF #Temporizador_Pos_Mistura.Q THEN

       #inOutControle.Pos_Mistura.Finalizado_Mistura := true;

   ELSE
       #inOutControle.Pos_Mistura.Finalizado_Mistura := false;
   END_IF;
END_REGION

REGION Network 6 (SCL): Transporte Pós Mistura Para Produto Acabado
   //Liberado Transportar
   IF NOT #inNivel_Superior_Silo_Produto_Acabado AND//Verifica se ainda tem espaço no silo através do nível alto
       #inOutControle.Pos_Mistura.Finalizado_Mistura //Finalizado pós mistura e pronto para transporte
   THEN

       #inOutControle.Transporte_Produto_Acabado.Liberado_Iniciar_Transporte := true;
   ELSE    
       #inOutControle.Transporte_Produto_Acabado.Liberado_Iniciar_Transporte := false;
   END_IF;

   //Liga transporte para produto acabado
   IF #inOutControle.Pos_Mistura.Finalizado_Mistura AND
       #inOutControle.Transporte_Produto_Acabado.Liberado_Iniciar_Transporte
   THEN
       #inOutControle.Transporte_Produto_Acabado.Ligar := true;
       #inOutControle.Pos_Mistura.Iniciado_Mistura := false;
   END_IF;

   //Desliga transporte para produto acabado
   #Temporizador_Finalizado_Transporte_Pos_Mistura(IN := (NOT #inNivel_Inferior_Pos_Mistura),
                                                   PT := t#10s);

   IF #Temporizador_Finalizado_Transporte_Pos_Mistura.Q THEN
       #inOutControle.Transporte_Produto_Acabado.Ligar := false;

   END_IF;

   //Verifica se esta ligado
   IF #inOutControle.Transporte_Produto_Acabado.Ligar AND
       "DB_Controle_Equip"."49".Aciona_Lado2 AND
       "DB_Controle_Equip"."62".ligado
   THEN
       #inOutControle.Transporte_Produto_Acabado.Ligado := true;
   ELSE
       #inOutControle.Transporte_Produto_Acabado.Ligado := false;
   END_IF;

   IF "DB_Controle_Equip"."62".Corrente_Atual <= "DB_Controle_Equip"."62".SP_Corrente_Motor_Vazio AND
       "DB_Controle_Equip"."62".ligado
   THEN
       #Elevador_62_Sem_Carga := true;
   ELSE
       #Elevador_62_Sem_Carga := false;
   END_IF;


   #Tempo_Transporte_Para_Produto_Acabado(IN := #Elevador_62_Sem_Carga,
                                          PT := t#5s);

   IF #Tempo_Transporte_Para_Produto_Acabado.Q AND
       NOT #inNivel_Inferior_Pos_Mistura AND
       #inOutControle.Transporte_Produto_Acabado.Ligado
   THEN
       #inOutControle.Transporte_Produto_Acabado.Ligar := false;

   END_IF;
END_REGION

REGION Network 7: Emergencia de processo
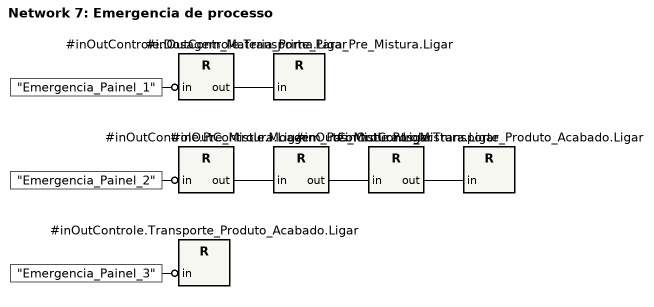
   IF NOT "Emergencia_Painel_1" THEN
       #inOutControle.Dosagem_Materia_Prima.Ligar := FALSE;
       #inOutControle.Transporte_Para_Pre_Mistura.Ligar := FALSE;
   END_IF;
   IF NOT "Emergencia_Painel_2" THEN
       #inOutControle.Pre_Mistura.Ligar := FALSE;
       #inOutControle.Moagem_Pos_Mistura.Ligar := FALSE;
       #inOutControle.Pos_Mistura.Ligar := FALSE;
       #inOutControle.Transporte_Produto_Acabado.Ligar := FALSE;
   END_IF;
   IF NOT "Emergencia_Painel_3" THEN #inOutControle.Transporte_Produto_Acabado.Ligar := FALSE; END_IF;
END_REGION

REGION Network 8: =========================================
END_REGION

REGION Network 9: Liga, Desliga - Dosagem Matéria Prima
END_REGION
END_FUNCTION_BLOCK

FUNCTION_BLOCK "Controle_Descarga_Atuador_Linear"   // FB6, FBD
{ S7_Optimized_Access := 'TRUE' }
VERSION : 0.1
   VAR_INPUT
      inValor_Dosar : Real;   // Valor para dosar
      inValor_Atual_Balanca : Real;   // Valor da balança
      inAbertura_Maxima_Atuador : Real;   // Abertura Máxima Atuador Linear
      inInicio_Reducao : Real;   // Valor de Inicio da redução
      inFechamento_Antecipado : Real;   // Fechar antecipadamente em um percentual especifico, como fechar a 3% do restante
      inDosar : Bool;   // Solicita dosar automatico
   END_VAR
   VAR_OUTPUT
      outPosicao_Atuador : Real;   // Posicao solicitada atuador
      outDosagem_Finalizada : Bool;   // Dosagem finalizada
      outDosagem_Iniciada : Bool;   // Dosagem iniciada
      outValor_Dosado_Ultima_Dosagem : Real;   // Valor dosado na ultima dosagem
   END_VAR
   VAR
      Valor_Tara_Balanca : Real;   // Tara capturada antes de iniciar a dosagem
      Tempo_Estabilizacao_Balanca : TON_TIME;
   END_VAR
   VAR_TEMP
      Valor_Atual_Balanca_Corrigido : Real;   // Valor atual da balança - tara
      Valor_Atual_Balanca_Percentual : Real;   // Valor atual da balança em percentual, de acordo com a dosagem solicitada
      Segunda_Reducao : Real;   // Percentual da segunda redução
      Terceira_Reducao : Real;   // Percentual da terceira redução
      Quarta_Reducao : Real;   // Percentual da quarta redução
      Quinta_Reducao : Real;   // Percentual da quinta redução
   END_VAR
BEGIN

REGION Network 1 (SCL): Tara capturada antes de iniciar a dosagem
   //Maycon Lutz
   //Sistema de redução para controle de dosagem
   //Funcionamento: Inicia a dosagem, é aberto o máximo do atuador, após atingir o inicio da redução
   //em percentual, é reduzido até fechar de acordo com as reduções abaixo
   //Reduções: São 5 reduções, exemplo considerando abertura máxima de 100% do atuador.
   //1 - 50% da abertura máxima = 50%
   //2 - 50% do resultado de 1 = 25%
   //3 - 50% do resultado de 2 = 12.5%
   //4 - 50% do resultado de 3 = 6,25%
   //5 - 50% do resultado de 4 = 3,125%
   //
   //Exemplo 1 de funcionamento:
   //Valor a dosar: 1000Kg
   //Valor atual: 0Kg
   //Abertura máxima: 100%
   //Fechamento antecipado: 2%
   //Inicio redução: 70% - 70 por cento de 1000 = inicio da redução 700Kg.
   //
   //500kg de valor atual = abertura de 100%
   //699kg de valor atual = abertura de 100%
   //700kg de valor atual = abertura de 50%
   //759kg de valor atual = abertura de 50%
   //760kg de valor atual = abertura de 25%
   //819kg de valor atual = abertura de 25%
   //820kg de valor atual = abertura de 12,5%
   //879kg de valor atual = abertura de 12,5%
   //880kg de valor atual = abertura de 6,25%
   //939kg de valor atual = abertura de 6,25%
   //940kg de valor atual = abertura de 3,125%
   //979kg de valor atual = abertura de 3,125%
   //980kg de valor atual = abertura de 0% - Fechamento antecipado entrou em ação
   //
   //70% = 700Kg - Primeira redução
   //76% = 760Kg - Segunda redução
   //82% = 820Kg - Terceira redução
   //88% = 880Kg - Quarta redução
   //94% = 940Kg - Quinta redução


   IF #inDosar THEN

       IF NOT #outDosagem_Iniciada THEN
           #Valor_Tara_Balanca := #inValor_Atual_Balanca;
           #outValor_Dosado_Ultima_Dosagem := 0;
           #outDosagem_Iniciada := true;
       ELSE
           #Valor_Atual_Balanca_Corrigido := #inValor_Atual_Balanca - #Valor_Tara_Balanca;

       END_IF;

       IF NOT #outDosagem_Finalizada THEN

           //Calcula valor atual em percentual da dosagem
           #Valor_Atual_Balanca_Percentual := (#Valor_Atual_Balanca_Corrigido / #inValor_Dosar) * 100;

           //verifica se o valor é menor do que o inicio da redução, se for começa as reduções
           //caso não assume valor máximo do atuador
           IF #Valor_Atual_Balanca_Percentual < #inInicio_Reducao THEN
               #outPosicao_Atuador := #inAbertura_Maxima_Atuador;
           ELSE
               #Tempo_Estabilizacao_Balanca(IN := #Valor_Atual_Balanca_Percentual >= 100,
                                            PT := t#5s);


               IF #Valor_Atual_Balanca_Percentual >= 100 THEN

                   IF #Tempo_Estabilizacao_Balanca.Q THEN
                       #outDosagem_Finalizada := true;
                   END_IF;

                   #outPosicao_Atuador := 0;
                   #outValor_Dosado_Ultima_Dosagem := #Valor_Atual_Balanca_Corrigido;

               ELSE     
                   IF #inFechamento_Antecipado >= (100 - #Valor_Atual_Balanca_Percentual) THEN
                       #outPosicao_Atuador := 0;
                   ELSE
                       //Calculo do percentual de cada redução
                       #Segunda_Reducao := (((100 - #inInicio_Reducao) / 5)) + #inInicio_Reducao;
                       #Terceira_Reducao := (((100 - #inInicio_Reducao) / 5) * 2) + #inInicio_Reducao;
                       #Quarta_Reducao := (((100 - #inInicio_Reducao) / 5) * 3) + #inInicio_Reducao;
                       #Quinta_Reducao := (((100 - #inInicio_Reducao) / 5) * 4) + #inInicio_Reducao;

                       IF #Valor_Atual_Balanca_Percentual < #Segunda_Reducao THEN //Primeira redução
                           #outPosicao_Atuador := #inAbertura_Maxima_Atuador / 2;
                       ELSIF #Valor_Atual_Balanca_Percentual < #Terceira_Reducao THEN//Segunda redução
                           #outPosicao_Atuador := (#inAbertura_Maxima_Atuador / 2) / 2;
                       ELSIF #Valor_Atual_Balanca_Percentual < #Quarta_Reducao THEN//Terceira redução
                           #outPosicao_Atuador := ((#inAbertura_Maxima_Atuador / 2) / 2) / 2;
                       ELSIF #Valor_Atual_Balanca_Percentual < #Quinta_Reducao THEN//Quarta redução
                           #outPosicao_Atuador := (((#inAbertura_Maxima_Atuador / 2) / 2) / 2) / 2;
                       ELSIF #Valor_Atual_Balanca_Percentual > #Quinta_Reducao THEN//Quinta redução
                           #outPosicao_Atuador := ((((#inAbertura_Maxima_Atuador / 2) / 2) / 2) / 2) / 2;
                       END_IF;
                   END_IF;
               END_IF;

           END_IF;
           #outValor_Dosado_Ultima_Dosagem := #Valor_Atual_Balanca_Corrigido;
       END_IF;
   ELSE
       #outPosicao_Atuador := 0;
       #outDosagem_Finalizada := false;
       #outDosagem_Iniciada := false;
   END_IF;
END_REGION
END_FUNCTION_BLOCK

